gfCNCPoint3[6064] = {X 169.2391, Y 33.2115, Z -3.8333, A 0.000, B 0.000, C 0.000 }
gfCNCPoint3[6065] = {X 169.6133, Y 31.4141, Z -3.8333, A 0.000, B 0.000, C 0.000 }
gfCNCPoint3[6066] = {X 170.2096, Y 29.6777, Z -3.8333, A 0.000, B 0.000, C 0.000 }
gfCNCPoint3[6067] = {X 170.8485, Y 28.3707, Z -3.8333, A 0.000, B 0.000, C 0.000 }
gfCNCPoint3[6068] = {X 171.6564, Y 27.1608, Z -3.8333, A 0.000, B 0.000, C 0.000 }
gfCNCPoint3[6069] = {X 172.6187, Y 26.0698, Z -3.8333, A 0.000, B 0.000, C 0.000 }
gfCNCPoint3[6070] = {X 173.7182, Y 25.1171, Z -3.8333, A 0.000, B 0.000, C 0.000 }
gfCNCPoint3[6071] = {X 174.9352, Y 24.3200, Z -3.8333, A 0.000, B 0.000, C 0.000 }
gfCNCPoint3[6072] = {X 174.1525, Y 23.9324, Z -3.8333, A 0.000, B 0.000, C 0.000 }
gfCNCPoint3[6073] = {X 173.4637, Y 23.3952, Z -3.8333, A 0.000, B 0.000, C 0.000 }
gfCNCPoint3[6074] = {X 172.8971, Y 22.7305, Z -3.8333, A 0.000, B 0.000, C 0.000 }
gfCNCPoint3[6075] = {X 172.4758, Y 21.9655, Z -3.8333, A 0.000, B 0.000, C 0.000 }
gfCNCPoint3[6076] = {X 171.1581, Y 18.7388, Z -3.8333, A 0.000, B 0.000, C 0.000 }
gfCNCPoint3[6077] = {X 167.4550, Y 20.2510, Z -3.8333, A 0.000, B 0.000, C 0.000 }
gfCNCPoint3[6078] = {X 171.2322, Y 18.7085, Z -3.8333, A 0.000, B 0.000, C 0.000 }
gfCNCPoint3[6079] = {X 169.9145, Y 15.4818, Z -3.8333, A 0.000, B 0.000, C 0.000 }
gfCNCPoint3[6080] = {X 169.6699, Y 14.6462, Z -3.8333, A 0.000, B 0.000, C 0.000 }
gfCNCPoint3[6081] = {X 169.6011, Y 13.7783, Z -3.8333, A 0.000, B 0.000, C 0.000 }
gfCNCPoint3[6082] = {X 169.7111, Y 12.9146, Z -3.8333, A 0.000, B 0.000, C 0.000 }
gfCNCPoint3[6083] = {X 169.9952, Y 12.0915, Z -3.8333, A 0.000, B 0.000, C 0.000 }
gfCNCPoint3[6084] = {X 170.4414, Y 11.3439, Z -3.8333, A 0.000, B 0.000, C 0.000 }
gfCNCPoint3[6085] = {X 171.0309, Y 10.7031, Z -3.8333, A 0.000, B 0.000, C 0.000 }
gfCNCPoint3[6086] = {X 171.7389, Y 10.1963, Z -3.8333, A 0.000, B 0.000, C 0.000 }
gfCNCPoint3[6087] = {X 172.3689, Y 9.8371, Z -3.8333, A 0.000, B 0.000, C 0.000 }
gfCNCPoint3[6088] = {X 173.2427, Y 9.4701, Z -3.8333, A 0.000, B 0.000, C 0.000 }
gfCNCPoint3[6089] = {X 174.1763, Y 9.3065, Z -3.8333, A 0.000, B 0.000, C 0.000 }
gfCNCPoint3[6090] = {X 175.1229, Y 9.3543, Z -3.8333, A 0.000, B 0.000, C 0.000 }
gfCNCPoint3[6091] = {X 176.0352, Y 9.6112, Z -3.8333, A 0.000, B 0.000, C 0.000 }
gfCNCPoint3[6092] = {X 178.2247, Y 8.6863, Z -3.8333, A 0.000, B 0.000, C 0.000 }
gfCNCPoint3[6093] = {X 180.4959, Y 7.9856, Z -3.8333, A 0.000, B 0.000, C 0.000 }
gfCNCPoint3[6094] = {X 182.8259, Y 7.5163, Z -3.8333, A 0.000, B 0.000, C 0.000 }
gfCNCPoint3[6095] = {X 185.1913, Y 7.2829, Z -3.8333, A 0.000, B 0.000, C 0.000 }
gfCNCPoint3[6096] = {X 187.5681, Y 7.2880, Z -3.8333, A 0.000, B 0.000, C 0.000 }
gfCNCPoint3[6097] = {X 189.9324, Y 7.5314, Z -3.8333, A 0.000, B 0.000, C 0.000 }
gfCNCPoint3[6098] = {X 191.6817, Y 7.8911, Z -3.8333, A 0.000, B 0.000, C 0.000 }
gfCNCPoint3[6099] = {X 193.3847, Y 8.4286, Z -3.8333, A 0.000, B 0.000, C 0.000 }
gfCNCPoint3[6100] = {X 195.0236, Y 9.1381, Z -3.8333, A 0.000, B 0.000, C 0.000 }
gfCNCPoint3[6101] = {X 196.5809, Y 10.0121, Z -3.8333, A 0.000, B 0.000, C 0.000 }
gfCNCPoint3[6102] = {X 198.0403, Y 11.0414, Z -3.8333, A 0.000, B 0.000, C 0.000 }
gfCNCPoint3[6103] = {X 199.3400, Y 12.2309, Z -3.8333, A 0.000, B 0.000, C 0.000 }
gfCNCPoint3[6104] = {X 200.4666, Y 13.5854, Z -3.8333, A 0.000, B 0.000, C 0.000 }
gfCNCPoint3[6105] = {X 201.3992, Y 15.0802, Z -3.8333, A 0.000, B 0.000, C 0.000 }
gfCNCPoint3[6106] = {X 202.1206, Y 16.6876, Z -3.8333, A 0.000, B 0.000, C 0.000 }
gfCNCPoint3[6107] = {X 202.5921, Y 18.3349, Z -3.8333, A 0.000, B 0.000, C 0.000 }
gfCNCPoint3[6108] = {X 202.8719, Y 20.0254, Z -3.8333, A 0.000, B 0.000, C 0.000 }
gfCNCPoint3[6109] = {X 202.9564, Y 21.7368, Z -3.8333, A 0.000, B 0.000, C 0.000 }
gfCNCPoint3[6110] = {X 202.8443, Y 23.4466, Z -3.8333, A 0.000, B 0.000, C 0.000 }
gfCNCPoint3[6111] = {X 202.5373, Y 25.1324, Z -3.8333, A 0.000, B 0.000, C 0.000 }
gfCNCPoint3[6112] = {X 202.0878, Y 26.5970, Z -3.8333, A 0.000, B 0.000, C 0.000 }
gfCNCPoint3[6113] = {X 201.4494, Y 27.9897, Z -3.8333, A 0.000, B 0.000, C 0.000 }
gfCNCPoint3[6114] = {X 200.6332, Y 29.2862, Z -3.8333, A 0.000, B 0.000, C 0.000 }
gfCNCPoint3[6115] = {X 199.6535, Y 30.4640, Z -3.8333, A 0.000, B 0.000, C 0.000 }
gfCNCPoint3[6116] = {X 198.5272, Y 31.5026, Z -3.8333, A 0.000, B 0.000, C 0.000 }
gfCNCPoint3[6117] = {X 199.3587, Y 31.8264, Z -3.8333, A 0.000, B 0.000, C 0.000 }
gfCNCPoint3[6118] = {X 200.1039, Y 32.3172, Z -3.8333, A 0.000, B 0.000, C 0.000 }
gfCNCPoint3[6119] = {X 200.7300, Y 32.9530, Z -3.8333, A 0.000, B 0.000, C 0.000 }
gfCNCPoint3[6120] = {X 201.2091, Y 33.7058, Z -3.8333, A 0.000, B 0.000, C 0.000 }
gfCNCPoint3[6121] = {X 204.2502, Y 39.9879, Z -3.8333, A 0.000, B 0.000, C 0.000 }
gfCNCPoint3[6122] = {X 204.5648, Y 40.8802, Z -3.8333, A 0.000, B 0.000, C 0.000 }
gfCNCPoint3[6123] = {X 204.6737, Y 41.8200, Z -3.8333, A 0.000, B 0.000, C 0.000 }
gfCNCPoint3[6124] = {X 204.5715, Y 42.7606, Z -3.8333, A 0.000, B 0.000, C 0.000 }
gfCNCPoint3[6125] = {X 204.2633, Y 43.6551, Z -3.8333, A 0.000, B 0.000, C 0.000 }
gfCNCPoint3[6126] = {X 203.7643, Y 44.4590, Z -3.8333, A 0.000, B 0.000, C 0.000 }
gfCNCPoint3[6127] = {X 203.0996, Y 45.1323, Z -3.8333, A 0.000, B 0.000, C 0.000 }
gfCNCPoint3[6128] = {X 202.5633, Y 45.5658, Z -3.8333, A 0.000, B 0.000, C 0.000 }
gfCNCPoint3[6129] = {X 201.8656, Y 46.0241, Z -3.8333, A 0.000, B 0.000, C 0.000 }
gfCNCPoint3[6130] = {X 201.0918, Y 46.3373, Z -3.8333, A 0.000, B 0.000, C 0.000 }
gfCNCPoint3[6131] = {X 200.2717, Y 46.4933, Z -3.8333, A 0.000, B 0.000, C 0.000 }
gfCNCPoint3[6132] = {X 199.4370, Y 46.4861, Z -3.8333, A 0.000, B 0.000, C 0.000 }
gfCNCPoint3[6133] = {X 198.6197, Y 46.3161, Z -3.8333, A 0.000, B 0.000, C 0.000 }
gfCNCPoint3[6134] = {X 196.8802, Y 47.2412, Z -3.8333, A 0.000, B 0.000, C 0.000 }
gfCNCPoint3[6135] = {X 195.0811, Y 48.0444, Z -3.8333, A 0.000, B 0.000, C 0.000 }
gfCNCPoint3[6136] = {X 193.2311, Y 48.7221, Z -3.8333, A 0.000, B 0.000, C 0.000 }
gfCNCPoint3[6137] = {X 191.3389, Y 49.2709, Z -3.8333, A 0.000, B 0.000, C 0.000 }
gfCNCPoint3[6138] = {X 189.4027, Y 49.6631, Z -3.8333, A 0.000, B 0.000, C 0.000 }
gfCNCPoint3[6139] = {X 187.4396, Y 49.8846, Z -3.8333, A 0.000, B 0.000, C 0.000 }
gfCNCPoint3[6140] = {X 185.4646, Y 49.9336, Z -3.8333, A 0.000, B 0.000, C 0.000 }
gfCNCPoint3[6141] = {X 183.4929, Y 49.8097, Z -3.8333, A 0.000, B 0.000, C 0.000 }
gfCNCPoint3[6142] = {X 181.5396, Y 49.5138, Z -3.8333, A 0.000, B 0.000, C 0.000 }
gfCNCPoint3[6143] = {X 179.6619, Y 49.0445, Z -3.8333, A 0.000, B 0.000, C 0.000 }
gfCNCPoint3[6144] = {X 177.8500, Y 48.3642, Z -3.8333, A 0.000, B 0.000, C 0.000 }
gfCNCPoint3[6145] = {X 176.1273, Y 47.4818, Z -3.8333, A 0.000, B 0.000, C 0.000 }
gfCNCPoint3[6146] = {X 174.5165, Y 46.4089, Z -3.8333, A 0.000, B 0.000, C 0.000 }
gfCNCPoint3[6147] = {X 173.2910, Y 45.3745, Z -3.8333, A 0.000, B 0.000, C 0.000 }
gfCNCPoint3[6148] = {X 172.2004, Y 44.1988, Z -3.8333, A 0.000, B 0.000, C 0.000 }
gfCNCPoint3[6149] = {X 171.2610, Y 42.8990, Z -3.8333, A 0.000, B 0.000, C 0.000 }
gfCNCPoint3[6150] = {X 170.4868, Y 41.4946, Z -3.8333, A 0.000, B 0.000, C 0.000 }
gfCNCPoint3[6151] = {X 169.8892, Y 40.0065, Z -3.8333, A 0.000, B 0.000, C 0.000 }
gfCNCPoint3[6152] = {X 169.4771, Y 38.4567, Z -3.8333, A 0.000, B 0.000, C 0.000 }
gfCNCPoint3[6153] = {X 169.2566, Y 36.8682, Z -3.8333, A 0.000, B 0.000, C 0.000 }
gfCNCPoint3[6154] = {X 169.1729, Y 35.0439, Z -3.8333, A 0.000, B 0.000, C 0.000 }
gfCNCPoint3[6155] = {X 169.3183, Y 33.2234, Z -3.8333, A 0.000, B 0.000, C 0.000 }
gfCNCPoint3[6156] = {X 169.6904, Y 31.4354, Z -3.8333, A 0.000, B 0.000, C 0.000 }
gfCNCPoint3[6157] = {X 170.2836, Y 29.7081, Z -3.8333, A 0.000, B 0.000, C 0.000 }
gfCNCPoint3[6158] = {X 170.9356, Y 28.3799, Z -3.8333, A 0.000, B 0.000, C 0.000 }
gfCNCPoint3[6159] = {X 171.7633, Y 27.1534, Z -3.8333, A 0.000, B 0.000, C 0.000 }
gfCNCPoint3[6160] = {X 172.7511, Y 26.0519, Z -3.8333, A 0.000, B 0.000, C 0.000 }
gfCNCPoint3[6161] = {X 173.8805, Y 25.0960, Z -3.8333, A 0.000, B 0.000, C 0.000 }
gfCNCPoint3[6162] = {X 175.1302, Y 24.3037, Z -3.8333, A 0.000, B 0.000, C 0.000 }
gfCNCPoint3[6163] = {X 174.3086, Y 23.9335, Z -3.8333, A 0.000, B 0.000, C 0.000 }
gfCNCPoint3[6164] = {X 173.5838, Y 23.3981, Z -3.8333, A 0.000, B 0.000, C 0.000 }
gfCNCPoint3[6165] = {X 172.9885, Y 22.7217, Z -3.8333, A 0.000, B 0.000, C 0.000 }
gfCNCPoint3[6166] = {X 172.5496, Y 21.9347, Z -3.8333, A 0.000, B 0.000, C 0.000 }
gfCNCPoint3[6167] = {X 171.2322, Y 18.7085, Z -3.8333, A 0.000, B 0.000, C 0.000 }
gfCNCPoint3[6168] = {X 167.5291, Y 20.2207, Z -3.8333, A 0.000, B 0.000, C 0.000 }
gfCNCPoint3[6169] = {X 171.3062, Y 18.6783, Z -3.8333, A 0.000, B 0.000, C 0.000 }
gfCNCPoint3[6170] = {X 169.9886, Y 15.4516, Z -3.8333, A 0.000, B 0.000, C 0.000 }
gfCNCPoint3[6171] = {X 169.7252, Y 14.4911, Z -3.8333, A 0.000, B 0.000, C 0.000 }
gfCNCPoint3[6172] = {X 169.6977, Y 13.4955, Z -3.8333, A 0.000, B 0.000, C 0.000 }
gfCNCPoint3[6173] = {X 169.9076, Y 12.5218, Z -3.8333, A 0.000, B 0.000, C 0.000 }
gfCNCPoint3[6174] = {X 170.3429, Y 11.6260, Z -3.8333, A 0.000, B 0.000, C 0.000 }
gfCNCPoint3[6175] = {X 170.9787, Y 10.8594, Z -3.8333, A 0.000, B 0.000, C 0.000 }
gfCNCPoint3[6176] = {X 171.7785, Y 10.2658, Z -3.8333, A 0.000, B 0.000, C 0.000 }
gfCNCPoint3[6177] = {X 172.4082, Y 9.9068, Z -3.8333, A 0.000, B 0.000, C 0.000 }
gfCNCPoint3[6178] = {X 173.2740, Y 9.5443, Z -3.8333, A 0.000, B 0.000, C 0.000 }
gfCNCPoint3[6179] = {X 174.1991, Y 9.3853, Z -3.8333, A 0.000, B 0.000, C 0.000 }
gfCNCPoint3[6180] = {X 175.1362, Y 9.4376, Z -3.8333, A 0.000, B 0.000, C 0.000 }
gfCNCPoint3[6181] = {X 176.0378, Y 9.6988, Z -3.8333, A 0.000, B 0.000, C 0.000 }
gfCNCPoint3[6182] = {X 178.2241, Y 8.7716, Z -3.8333, A 0.000, B 0.000, C 0.000 }
gfCNCPoint3[6183] = {X 180.4925, Y 8.0690, Z -3.8333, A 0.000, B 0.000, C 0.000 }
gfCNCPoint3[6184] = {X 182.8201, Y 7.5980, Z -3.8333, A 0.000, B 0.000, C 0.000 }
gfCNCPoint3[6185] = {X 185.1832, Y 7.3634, Z -3.8333, A 0.000, B 0.000, C 0.000 }
gfCNCPoint3[6186] = {X 187.5580, Y 7.3676, Z -3.8333, A 0.000, B 0.000, C 0.000 }
gfCNCPoint3[6187] = {X 189.9203, Y 7.6105, Z -3.8333, A 0.000, B 0.000, C 0.000 }
gfCNCPoint3[6188] = {X 191.6615, Y 7.9685, Z -3.8333, A 0.000, B 0.000, C 0.000 }
gfCNCPoint3[6189] = {X 193.3567, Y 8.5035, Z -3.8333, A 0.000, B 0.000, C 0.000 }
gfCNCPoint3[6190] = {X 194.9880, Y 9.2097, Z -3.8333, A 0.000, B 0.000, C 0.000 }
gfCNCPoint3[6191] = {X 196.5382, Y 10.0797, Z -3.8333, A 0.000, B 0.000, C 0.000 }
gfCNCPoint3[6192] = {X 197.9908, Y 11.1044, Z -3.8333, A 0.000, B 0.000, C 0.000 }
gfCNCPoint3[6193] = {X 199.2823, Y 12.2863, Z -3.8333, A 0.000, B 0.000, C 0.000 }
gfCNCPoint3[6194] = {X 200.4017, Y 13.6323, Z -3.8333, A 0.000, B 0.000, C 0.000 }
gfCNCPoint3[6195] = {X 201.3284, Y 15.1175, Z -3.8333, A 0.000, B 0.000, C 0.000 }
gfCNCPoint3[6196] = {X 202.0453, Y 16.7146, Z -3.8333, A 0.000, B 0.000, C 0.000 }
gfCNCPoint3[6197] = {X 202.5142, Y 18.3531, Z -3.8333, A 0.000, B 0.000, C 0.000 }
gfCNCPoint3[6198] = {X 202.7924, Y 20.0344, Z -3.8333, A 0.000, B 0.000, C 0.000 }
gfCNCPoint3[6199] = {X 202.8764, Y 21.7366, Z -3.8333, A 0.000, B 0.000, C 0.000 }
gfCNCPoint3[6200] = {X 202.7649, Y 23.4371, Z -3.8333, A 0.000, B 0.000, C 0.000 }
gfCNCPoint3[6201] = {X 202.4595, Y 25.1138, Z -3.8333, A 0.000, B 0.000, C 0.000 }
gfCNCPoint3[6202] = {X 202.0016, Y 26.5984, Z -3.8333, A 0.000, B 0.000, C 0.000 }
gfCNCPoint3[6203] = {X 201.3483, Y 28.0081, Z -3.8333, A 0.000, B 0.000, C 0.000 }
gfCNCPoint3[6204] = {X 200.5114, Y 29.3171, Z -3.8333, A 0.000, B 0.000, C 0.000 }
gfCNCPoint3[6205] = {X 199.5062, Y 30.5018, Z -3.8333, A 0.000, B 0.000, C 0.000 }
gfCNCPoint3[6206] = {X 198.3508, Y 31.5406, Z -3.8333, A 0.000, B 0.000, C 0.000 }
gfCNCPoint3[6207] = {X 199.2144, Y 31.8439, Z -3.8333, A 0.000, B 0.000, C 0.000 }
gfCNCPoint3[6208] = {X 199.9908, Y 32.3287, Z -3.8333, A 0.000, B 0.000, C 0.000 }
gfCNCPoint3[6209] = {X 200.6423, Y 32.9716, Z -3.8333, A 0.000, B 0.000, C 0.000 }
gfCNCPoint3[6210] = {X 201.1375, Y 33.7414, Z -3.8333, A 0.000, B 0.000, C 0.000 }
gfCNCPoint3[6211] = {X 204.1781, Y 40.0227, Z -3.8333, A 0.000, B 0.000, C 0.000 }
gfCNCPoint3[6212] = {X 204.4868, Y 40.8982, Z -3.8333, A 0.000, B 0.000, C 0.000 }
gfCNCPoint3[6213] = {X 204.5937, Y 41.8203, Z -3.8333, A 0.000, B 0.000, C 0.000 }
gfCNCPoint3[6214] = {X 204.4934, Y 42.7431, Z -3.8333, A 0.000, B 0.000, C 0.000 }
gfCNCPoint3[6215] = {X 204.1910, Y 43.6208, Z -3.8333, A 0.000, B 0.000, C 0.000 }
gfCNCPoint3[6216] = {X 203.7015, Y 44.4095, Z -3.8333, A 0.000, B 0.000, C 0.000 }
gfCNCPoint3[6217] = {X 203.0493, Y 45.0700, Z -3.8333, A 0.000, B 0.000, C 0.000 }
gfCNCPoint3[6218] = {X 202.5131, Y 45.5036, Z -3.8333, A 0.000, B 0.000, C 0.000 }
gfCNCPoint3[6219] = {X 201.8223, Y 45.9565, Z -3.8333, A 0.000, B 0.000, C 0.000 }
gfCNCPoint3[6220] = {X 201.0558, Y 46.2645, Z -3.8333, A 0.000, B 0.000, C 0.000 }
gfCNCPoint3[6221] = {X 200.2436, Y 46.4154, Z -3.8333, A 0.000, B 0.000, C 0.000 }
gfCNCPoint3[6222] = {X 199.4177, Y 46.4035, Z -3.8333, A 0.000, B 0.000, C 0.000 }
gfCNCPoint3[6223] = {X 198.6103, Y 46.2291, Z -3.8333, A 0.000, B 0.000, C 0.000 }
gfCNCPoint3[6224] = {X 196.8688, Y 47.1577, Z -3.8333, A 0.000, B 0.000, C 0.000 }
gfCNCPoint3[6225] = {X 195.0674, Y 47.9637, Z -3.8333, A 0.000, B 0.000, C 0.000 }
gfCNCPoint3[6226] = {X 193.2146, Y 48.6433, Z -3.8333, A 0.000, B 0.000, C 0.000 }
gfCNCPoint3[6227] = {X 191.3193, Y 49.1933, Z -3.8333, A 0.000, B 0.000, C 0.000 }
gfCNCPoint3[6228] = {X 189.3899, Y 49.5842, Z -3.8333, A 0.000, B 0.000, C 0.000 }
gfCNCPoint3[6229] = {X 187.4338, Y 49.8048, Z -3.8333, A 0.000, B 0.000, C 0.000 }
gfCNCPoint3[6230] = {X 185.4659, Y 49.8536, Z -3.8333, A 0.000, B 0.000, C 0.000 }
gfCNCPoint3[6231] = {X 183.5012, Y 49.7301, Z -3.8333, A 0.000, B 0.000, C 0.000 }
gfCNCPoint3[6232] = {X 181.5549, Y 49.4353, Z -3.8333, A 0.000, B 0.000, C 0.000 }
gfCNCPoint3[6233] = {X 179.6859, Y 48.9682, Z -3.8333, A 0.000, B 0.000, C 0.000 }
gfCNCPoint3[6234] = {X 177.8824, Y 48.2911, Z -3.8333, A 0.000, B 0.000, C 0.000 }
gfCNCPoint3[6235] = {X 176.1678, Y 47.4128, Z -3.8333, A 0.000, B 0.000, C 0.000 }
gfCNCPoint3[6236] = {X 174.5644, Y 46.3449, Z -3.8333, A 0.000, B 0.000, C 0.000 }
gfCNCPoint3[6237] = {X 173.3462, Y 45.3167, Z -3.8333, A 0.000, B 0.000, C 0.000 }
gfCNCPoint3[6238] = {X 172.2622, Y 44.1479, Z -3.8333, A 0.000, B 0.000, C 0.000 }
gfCNCPoint3[6239] = {X 171.3284, Y 42.8559, Z -3.8333, A 0.000, B 0.000, C 0.000 }
gfCNCPoint3[6240] = {X 170.5588, Y 41.4598, Z -3.8333, A 0.000, B 0.000, C 0.000 }
gfCNCPoint3[6241] = {X 169.9648, Y 39.9804, Z -3.8333, A 0.000, B 0.000, C 0.000 }
gfCNCPoint3[6242] = {X 169.5553, Y 38.4398, Z -3.8333, A 0.000, B 0.000, C 0.000 }
gfCNCPoint3[6243] = {X 169.3363, Y 36.8608, Z -3.8333, A 0.000, B 0.000, C 0.000 }
gfCNCPoint3[6244] = {X 169.2528, Y 35.0461, Z -3.8333, A 0.000, B 0.000, C 0.000 }
gfCNCPoint3[6245] = {X 169.3974, Y 33.2352, Z -3.8333, A 0.000, B 0.000, C 0.000 }
gfCNCPoint3[6246] = {X 169.7675, Y 31.4567, Z -3.8333, A 0.000, B 0.000, C 0.000 }
gfCNCPoint3[6247] = {X 170.3575, Y 29.7386, Z -3.8333, A 0.000, B 0.000, C 0.000 }
gfCNCPoint3[6248] = {X 171.0242, Y 28.3867, Z -3.8333, A 0.000, B 0.000, C 0.000 }
gfCNCPoint3[6249] = {X 171.8741, Y 27.1419, Z -3.8333, A 0.000, B 0.000, C 0.000 }
gfCNCPoint3[6250] = {X 172.8906, Y 26.0288, Z -3.8333, A 0.000, B 0.000, C 0.000 }
gfCNCPoint3[6251] = {X 174.0533, Y 25.0696, Z -3.8333, A 0.000, B 0.000, C 0.000 }
gfCNCPoint3[6252] = {X 175.3393, Y 24.2834, Z -3.8333, A 0.000, B 0.000, C 0.000 }
gfCNCPoint3[6253] = {X 174.4750, Y 23.9353, Z -3.8333, A 0.000, B 0.000, C 0.000 }
gfCNCPoint3[6254] = {X 173.7098, Y 23.4037, Z -3.8333, A 0.000, B 0.000, C 0.000 }
gfCNCPoint3[6255] = {X 173.0821, Y 22.7150, Z -3.8333, A 0.000, B 0.000, C 0.000 }
gfCNCPoint3[6256] = {X 172.6235, Y 21.9039, Z -3.8333, A 0.000, B 0.000, C 0.000 }
gfCNCPoint3[6257] = {X 171.3062, Y 18.6783, Z -3.8333, A 0.000, B 0.000, C 0.000 }
gfCNCPoint3[6258] = {X 167.6031, Y 20.1905, Z -3.8333, A 0.000, B 0.000, C 0.000 }
gfCNCPoint3[6259] = {X 171.3803, Y 18.6480, Z -3.8333, A 0.000, B 0.000, C 0.000 }
gfCNCPoint3[6260] = {X 170.0626, Y 15.4213, Z -3.8333, A 0.000, B 0.000, C 0.000 }
gfCNCPoint3[6261] = {X 169.8043, Y 14.4793, Z -3.8333, A 0.000, B 0.000, C 0.000 }
gfCNCPoint3[6262] = {X 169.7773, Y 13.5028, Z -3.8333, A 0.000, B 0.000, C 0.000 }
gfCNCPoint3[6263] = {X 169.9832, Y 12.5479, Z -3.8333, A 0.000, B 0.000, C 0.000 }
gfCNCPoint3[6264] = {X 170.4102, Y 11.6694, Z -3.8333, A 0.000, B 0.000, C 0.000 }
gfCNCPoint3[6265] = {X 171.0337, Y 10.9174, Z -3.8333, A 0.000, B 0.000, C 0.000 }
gfCNCPoint3[6266] = {X 171.8181, Y 10.3353, Z -3.8333, A 0.000, B 0.000, C 0.000 }
gfCNCPoint3[6267] = {X 172.4475, Y 9.9764, Z -3.8333, A 0.000, B 0.000, C 0.000 }
gfCNCPoint3[6268] = {X 173.3053, Y 9.6186, Z -3.8333, A 0.000, B 0.000, C 0.000 }
gfCNCPoint3[6269] = {X 174.2218, Y 9.4641, Z -3.8333, A 0.000, B 0.000, C 0.000 }
gfCNCPoint3[6270] = {X 175.1494, Y 9.5211, Z -3.8333, A 0.000, B 0.000, C 0.000 }
gfCNCPoint3[6271] = {X 176.0401, Y 9.7866, Z -3.8333, A 0.000, B 0.000, C 0.000 }
gfCNCPoint3[6272] = {X 178.2232, Y 8.8572, Z -3.8333, A 0.000, B 0.000, C 0.000 }
gfCNCPoint3[6273] = {X 180.4889, Y 8.1525, Z -3.8333, A 0.000, B 0.000, C 0.000 }
gfCNCPoint3[6274] = {X 182.8141, Y 7.6798, Z -3.8333, A 0.000, B 0.000, C 0.000 }
gfCNCPoint3[6275] = {X 185.1750, Y 7.4439, Z -3.8333, A 0.000, B 0.000, C 0.000 }
gfCNCPoint3[6276] = {X 187.5478, Y 7.4472, Z -3.8333, A 0.000, B 0.000, C 0.000 }
gfCNCPoint3[6277] = {X 189.9081, Y 7.6895, Z -3.8333, A 0.000, B 0.000, C 0.000 }
gfCNCPoint3[6278] = {X 191.6413, Y 8.0459, Z -3.8333, A 0.000, B 0.000, C 0.000 }
gfCNCPoint3[6279] = {X 193.3287, Y 8.5784, Z -3.8333, A 0.000, B 0.000, C 0.000 }
gfCNCPoint3[6280] = {X 194.9525, Y 9.2814, Z -3.8333, A 0.000, B 0.000, C 0.000 }
gfCNCPoint3[6281] = {X 196.4955, Y 10.1474, Z -3.8333, A 0.000, B 0.000, C 0.000 }
gfCNCPoint3[6282] = {X 197.9414, Y 11.1673, Z -3.8333, A 0.000, B 0.000, C 0.000 }
gfCNCPoint3[6283] = {X 199.2246, Y 12.3417, Z -3.8333, A 0.000, B 0.000, C 0.000 }
gfCNCPoint3[6284] = {X 200.3368, Y 13.6791, Z -3.8333, A 0.000, B 0.000, C 0.000 }
gfCNCPoint3[6285] = {X 201.2577, Y 15.1548, Z -3.8333, A 0.000, B 0.000, C 0.000 }
gfCNCPoint3[6286] = {X 201.9701, Y 16.7417, Z -3.8333, A 0.000, B 0.000, C 0.000 }
gfCNCPoint3[6287] = {X 202.4363, Y 18.3712, Z -3.8333, A 0.000, B 0.000, C 0.000 }
gfCNCPoint3[6288] = {X 202.7129, Y 20.0435, Z -3.8333, A 0.000, B 0.000, C 0.000 }
gfCNCPoint3[6289] = {X 202.7964, Y 21.7363, Z -3.8333, A 0.000, B 0.000, C 0.000 }
gfCNCPoint3[6290] = {X 202.6855, Y 23.4277, Z -3.8333, A 0.000, B 0.000, C 0.000 }
gfCNCPoint3[6291] = {X 202.3817, Y 25.0952, Z -3.8333, A 0.000, B 0.000, C 0.000 }
gfCNCPoint3[6292] = {X 201.9145, Y 26.6019, Z -3.8333, A 0.000, B 0.000, C 0.000 }
gfCNCPoint3[6293] = {X 201.2448, Y 28.0301, Z -3.8333, A 0.000, B 0.000, C 0.000 }
gfCNCPoint3[6294] = {X 200.3851, Y 29.3527, Z -3.8333, A 0.000, B 0.000, C 0.000 }
gfCNCPoint3[6295] = {X 199.3518, Y 30.5447, Z -3.8333, A 0.000, B 0.000, C 0.000 }
gfCNCPoint3[6296] = {X 198.1646, Y 31.5833, Z -3.8333, A 0.000, B 0.000, C 0.000 }
gfCNCPoint3[6297] = {X 199.0626, Y 31.8620, Z -3.8333, A 0.000, B 0.000, C 0.000 }
gfCNCPoint3[6298] = {X 199.8730, Y 32.3388, Z -3.8333, A 0.000, B 0.000, C 0.000 }
gfCNCPoint3[6299] = {X 200.5528, Y 32.9886, Z -3.8333, A 0.000, B 0.000, C 0.000 }
gfCNCPoint3[6300] = {X 201.0657, Y 33.7766, Z -3.8333, A 0.000, B 0.000, C 0.000 }
gfCNCPoint3[6301] = {X 204.1061, Y 40.0576, Z -3.8333, A 0.000, B 0.000, C 0.000 }
gfCNCPoint3[6302] = {X 204.4089, Y 40.9162, Z -3.8333, A 0.000, B 0.000, C 0.000 }
gfCNCPoint3[6303] = {X 204.5137, Y 41.8206, Z -3.8333, A 0.000, B 0.000, C 0.000 }
gfCNCPoint3[6304] = {X 204.4154, Y 42.7257, Z -3.8333, A 0.000, B 0.000, C 0.000 }
gfCNCPoint3[6305] = {X 204.1188, Y 43.5864, Z -3.8333, A 0.000, B 0.000, C 0.000 }
gfCNCPoint3[6306] = {X 203.6387, Y 44.3600, Z -3.8333, A 0.000, B 0.000, C 0.000 }
gfCNCPoint3[6307] = {X 202.9990, Y 45.0078, Z -3.8333, A 0.000, B 0.000, C 0.000 }
gfCNCPoint3[6308] = {X 202.4628, Y 45.4414, Z -3.8333, A 0.000, B 0.000, C 0.000 }
gfCNCPoint3[6309] = {X 201.7789, Y 45.8889, Z -3.8333, A 0.000, B 0.000, C 0.000 }
gfCNCPoint3[6310] = {X 201.0198, Y 46.1916, Z -3.8333, A 0.000, B 0.000, C 0.000 }
gfCNCPoint3[6311] = {X 200.2157, Y 46.3375, Z -3.8333, A 0.000, B 0.000, C 0.000 }
gfCNCPoint3[6312] = {X 199.3986, Y 46.3207, Z -3.8333, A 0.000, B 0.000, C 0.000 }
gfCNCPoint3[6313] = {X 198.6011, Y 46.1420, Z -3.8333, A 0.000, B 0.000, C 0.000 }
gfCNCPoint3[6314] = {X 196.8577, Y 47.0740, Z -3.8333, A 0.000, B 0.000, C 0.000 }
gfCNCPoint3[6315] = {X 195.0538, Y 47.8828, Z -3.8333, A 0.000, B 0.000, C 0.000 }
gfCNCPoint3[6316] = {X 193.1981, Y 48.5645, Z -3.8333, A 0.000, B 0.000, C 0.000 }
gfCNCPoint3[6317] = {X 191.2996, Y 49.1157, Z -3.8333, A 0.000, B 0.000, C 0.000 }
gfCNCPoint3[6318] = {X 189.3772, Y 49.5052, Z -3.8333, A 0.000, B 0.000, C 0.000 }
gfCNCPoint3[6319] = {X 187.4280, Y 49.7250, Z -3.8333, A 0.000, B 0.000, C 0.000 }
gfCNCPoint3[6320] = {X 185.4671, Y 49.7736, Z -3.8333, A 0.000, B 0.000, C 0.000 }
gfCNCPoint3[6321] = {X 183.5094, Y 49.6505, Z -3.8333, A 0.000, B 0.000, C 0.000 }
gfCNCPoint3[6322] = {X 181.5701, Y 49.3567, Z -3.8333, A 0.000, B 0.000, C 0.000 }
gfCNCPoint3[6323] = {X 179.7099, Y 48.8918, Z -3.8333, A 0.000, B 0.000, C 0.000 }
gfCNCPoint3[6324] = {X 177.9148, Y 48.2179, Z -3.8333, A 0.000, B 0.000, C 0.000 }
gfCNCPoint3[6325] = {X 176.2082, Y 47.3438, Z -3.8333, A 0.000, B 0.000, C 0.000 }
gfCNCPoint3[6326] = {X 174.6124, Y 46.2809, Z -3.8333, A 0.000, B 0.000, C 0.000 }
gfCNCPoint3[6327] = {X 173.4015, Y 45.2588, Z -3.8333, A 0.000, B 0.000, C 0.000 }
gfCNCPoint3[6328] = {X 172.3239, Y 44.0970, Z -3.8333, A 0.000, B 0.000, C 0.000 }
gfCNCPoint3[6329] = {X 171.3958, Y 42.8127, Z -3.8333, A 0.000, B 0.000, C 0.000 }
gfCNCPoint3[6330] = {X 170.6308, Y 41.4249, Z -3.8333, A 0.000, B 0.000, C 0.000 }
gfCNCPoint3[6331] = {X 170.0405, Y 39.9544, Z -3.8333, A 0.000, B 0.000, C 0.000 }
gfCNCPoint3[6332] = {X 169.6335, Y 38.4230, Z -3.8333, A 0.000, B 0.000, C 0.000 }
gfCNCPoint3[6333] = {X 169.4159, Y 36.8534, Z -3.8333, A 0.000, B 0.000, C 0.000 }
gfCNCPoint3[6334] = {X 169.3328, Y 35.0483, Z -3.8333, A 0.000, B 0.000, C 0.000 }
gfCNCPoint3[6335] = {X 169.4765, Y 33.2471, Z -3.8333, A 0.000, B 0.000, C 0.000 }
gfCNCPoint3[6336] = {X 169.8447, Y 31.4780, Z -3.8333, A 0.000, B 0.000, C 0.000 }
gfCNCPoint3[6337] = {X 170.4315, Y 29.7690, Z -3.8333, A 0.000, B 0.000, C 0.000 }
gfCNCPoint3[6338] = {X 171.1148, Y 28.3902, Z -3.8333, A 0.000, B 0.000, C 0.000 }
gfCNCPoint3[6339] = {X 171.9902, Y 27.1247, Z -3.8333, A 0.000, B 0.000, C 0.000 }
gfCNCPoint3[6340] = {X 173.0392, Y 25.9989, Z -3.8333, A 0.000, B 0.000, C 0.000 }
gfCNCPoint3[6341] = {X 174.2400, Y 25.0365, Z -3.8333, A 0.000, B 0.000, C 0.000 }
gfCNCPoint3[6342] = {X 175.5672, Y 24.2578, Z -3.8333, A 0.000, B 0.000, C 0.000 }
gfCNCPoint3[6343] = {X 174.6550, Y 23.9381, Z -3.8333, A 0.000, B 0.000, C 0.000 }
gfCNCPoint3[6344] = {X 173.8437, Y 23.4127, Z -3.8333, A 0.000, B 0.000, C 0.000 }
gfCNCPoint3[6345] = {X 173.1787, Y 22.7113, Z -3.8333, A 0.000, B 0.000, C 0.000 }
gfCNCPoint3[6346] = {X 172.6973, Y 21.8731, Z -3.8333, A 0.000, B 0.000, C 0.000 }
gfCNCPoint3[6347] = {X 171.3803, Y 18.6480, Z -3.8333, A 0.000, B 0.000, C 0.000 }
gfCNCPoint3[6348] = {X 167.6770, Y 20.1603, Z -3.8333, A 0.000, B 0.000, C 0.000 }
gfCNCPoint3[6349] = {X 167.6769, Y 20.1601, Z -3.8333, A 0.000, B 0.000, C 0.000 }
gfCNCPoint3[6350] = {X 171.4542, Y 18.6179, Z -3.8333, A 0.000, B 0.000, C 0.000 }
gfCNCPoint3[6351] = {X 170.1367, Y 15.3911, Z -3.8333, A 0.000, B 0.000, C 0.000 }
gfCNCPoint3[6352] = {X 169.8835, Y 14.4675, Z -3.8333, A 0.000, B 0.000, C 0.000 }
gfCNCPoint3[6353] = {X 169.8570, Y 13.5102, Z -3.8333, A 0.000, B 0.000, C 0.000 }
gfCNCPoint3[6354] = {X 170.0588, Y 12.5740, Z -3.8333, A 0.000, B 0.000, C 0.000 }
gfCNCPoint3[6355] = {X 170.4774, Y 11.7127, Z -3.8333, A 0.000, B 0.000, C 0.000 }
gfCNCPoint3[6356] = {X 171.0888, Y 10.9755, Z -3.8333, A 0.000, B 0.000, C 0.000 }
gfCNCPoint3[6357] = {X 171.8578, Y 10.4048, Z -3.8333, A 0.000, B 0.000, C 0.000 }
gfCNCPoint3[6358] = {X 172.4867, Y 10.0462, Z -3.8333, A 0.000, B 0.000, C 0.000 }
gfCNCPoint3[6359] = {X 173.3363, Y 9.6929, Z -3.8333, A 0.000, B 0.000, C 0.000 }
gfCNCPoint3[6360] = {X 174.2443, Y 9.5431, Z -3.8333, A 0.000, B 0.000, C 0.000 }
gfCNCPoint3[6361] = {X 175.1624, Y 9.6048, Z -3.8333, A 0.000, B 0.000, C 0.000 }
gfCNCPoint3[6362] = {X 176.0421, Y 9.8746, Z -3.8333, A 0.000, B 0.000, C 0.000 }
gfCNCPoint3[6363] = {X 177.9051, Y 9.0624, Z -3.8333, A 0.000, B 0.000, C 0.000 }
gfCNCPoint3[6364] = {X 179.8314, Y 8.4146, Z -3.8333, A 0.000, B 0.000, C 0.000 }
gfCNCPoint3[6365] = {X 181.8066, Y 7.9362, Z -3.8333, A 0.000, B 0.000, C 0.000 }
gfCNCPoint3[6366] = {X 183.8158, Y 7.6308, Z -3.8333, A 0.000, B 0.000, C 0.000 }
gfCNCPoint3[6367] = {X 185.8440, Y 7.5006, Z -3.8333, A 0.000, B 0.000, C 0.000 }
gfCNCPoint3[6368] = {X 187.8758, Y 7.5467, Z -3.8333, A 0.000, B 0.000, C 0.000 }
gfCNCPoint3[6369] = {X 189.8959, Y 7.7686, Z -3.8333, A 0.000, B 0.000, C 0.000 }
gfCNCPoint3[6370] = {X 191.6211, Y 8.1233, Z -3.8333, A 0.000, B 0.000, C 0.000 }
gfCNCPoint3[6371] = {X 193.3006, Y 8.6533, Z -3.8333, A 0.000, B 0.000, C 0.000 }
gfCNCPoint3[6372] = {X 194.9169, Y 9.3530, Z -3.8333, A 0.000, B 0.000, C 0.000 }
gfCNCPoint3[6373] = {X 196.4528, Y 10.2150, Z -3.8333, A 0.000, B 0.000, C 0.000 }
gfCNCPoint3[6374] = {X 197.8920, Y 11.2302, Z -3.8333, A 0.000, B 0.000, C 0.000 }
gfCNCPoint3[6375] = {X 199.1669, Y 12.3971, Z -3.8333, A 0.000, B 0.000, C 0.000 }
gfCNCPoint3[6376] = {X 200.2720, Y 13.7259, Z -3.8333, A 0.000, B 0.000, C 0.000 }
gfCNCPoint3[6377] = {X 201.1869, Y 15.1921, Z -3.8333, A 0.000, B 0.000, C 0.000 }
gfCNCPoint3[6378] = {X 201.8948, Y 16.7687, Z -3.8333, A 0.000, B 0.000, C 0.000 }
gfCNCPoint3[6379] = {X 202.3584, Y 18.3894, Z -3.8333, A 0.000, B 0.000, C 0.000 }
gfCNCPoint3[6380] = {X 202.6334, Y 20.0525, Z -3.8333, A 0.000, B 0.000, C 0.000 }
gfCNCPoint3[6381] = {X 202.7164, Y 21.7361, Z -3.8333, A 0.000, B 0.000, C 0.000 }
gfCNCPoint3[6382] = {X 202.6060, Y 23.4182, Z -3.8333, A 0.000, B 0.000, C 0.000 }
gfCNCPoint3[6383] = {X 202.3039, Y 25.0766, Z -3.8333, A 0.000, B 0.000, C 0.000 }
gfCNCPoint3[6384] = {X 201.8264, Y 26.6077, Z -3.8333, A 0.000, B 0.000, C 0.000 }
gfCNCPoint3[6385] = {X 201.1382, Y 28.0565, Z -3.8333, A 0.000, B 0.000, C 0.000 }
gfCNCPoint3[6386] = {X 200.2531, Y 29.3941, Z -3.8333, A 0.000, B 0.000, C 0.000 }
gfCNCPoint3[6387] = {X 199.1886, Y 30.5938, Z -3.8333, A 0.000, B 0.000, C 0.000 }
gfCNCPoint3[6388] = {X 197.9659, Y 31.6319, Z -3.8333, A 0.000, B 0.000, C 0.000 }
gfCNCPoint3[6389] = {X 198.7277, Y 31.8158, Z -3.8333, A 0.000, B 0.000, C 0.000 }
gfCNCPoint3[6390] = {X 199.4391, Y 32.1448, Z -3.8333, A 0.000, B 0.000, C 0.000 }
gfCNCPoint3[6391] = {X 200.0726, Y 32.6061, Z -3.8333, A 0.000, B 0.000, C 0.000 }
gfCNCPoint3[6392] = {X 200.6040, Y 33.1821, Z -3.8333, A 0.000, B 0.000, C 0.000 }
gfCNCPoint3[6393] = {X 201.0129, Y 33.8507, Z -3.8333, A 0.000, B 0.000, C 0.000 }
gfCNCPoint3[6394] = {X 204.0341, Y 40.0925, Z -3.8333, A 0.000, B 0.000, C 0.000 }
gfCNCPoint3[6395] = {X 204.3309, Y 40.9342, Z -3.8333, A 0.000, B 0.000, C 0.000 }
gfCNCPoint3[6396] = {X 204.4337, Y 41.8209, Z -3.8333, A 0.000, B 0.000, C 0.000 }
gfCNCPoint3[6397] = {X 204.3373, Y 42.7082, Z -3.8333, A 0.000, B 0.000, C 0.000 }
gfCNCPoint3[6398] = {X 204.0465, Y 43.5521, Z -3.8333, A 0.000, B 0.000, C 0.000 }
gfCNCPoint3[6399] = {X 203.5758, Y 44.3105, Z -3.8333, A 0.000, B 0.000, C 0.000 }
gfCNCPoint3[6400] = {X 202.9487, Y 44.9456, Z -3.8333, A 0.000, B 0.000, C 0.000 }
gfCNCPoint3[6401] = {X 202.4125, Y 45.3791, Z -3.8333, A 0.000, B 0.000, C 0.000 }
gfCNCPoint3[6402] = {X 201.7357, Y 45.8212, Z -3.8333, A 0.000, B 0.000, C 0.000 }
gfCNCPoint3[6403] = {X 200.9839, Y 46.1186, Z -3.8333, A 0.000, B 0.000, C 0.000 }
gfCNCPoint3[6404] = {X 200.1879, Y 46.2594, Z -3.8333, A 0.000, B 0.000, C 0.000 }
gfCNCPoint3[6405] = {X 199.3797, Y 46.2377, Z -3.8333, A 0.000, B 0.000, C 0.000 }
gfCNCPoint3[6406] = {X 198.5923, Y 46.0546, Z -3.8333, A 0.000, B 0.000, C 0.000 }
gfCNCPoint3[6407] = {X 196.8468, Y 46.9902, Z -3.8333, A 0.000, B 0.000, C 0.000 }
gfCNCPoint3[6408] = {X 195.0404, Y 47.8019, Z -3.8333, A 0.000, B 0.000, C 0.000 }
gfCNCPoint3[6409] = {X 193.1818, Y 48.4857, Z -3.8333, A 0.000, B 0.000, C 0.000 }
gfCNCPoint3[6410] = {X 191.2800, Y 49.0382, Z -3.8333, A 0.000, B 0.000, C 0.000 }
gfCNCPoint3[6411] = {X 189.3644, Y 49.4262, Z -3.8333, A 0.000, B 0.000, C 0.000 }
gfCNCPoint3[6412] = {X 187.4222, Y 49.6453, Z -3.8333, A 0.000, B 0.000, C 0.000 }
gfCNCPoint3[6413] = {X 185.4683, Y 49.6936, Z -3.8333, A 0.000, B 0.000, C 0.000 }
gfCNCPoint3[6414] = {X 183.5177, Y 49.5710, Z -3.8333, A 0.000, B 0.000, C 0.000 }
gfCNCPoint3[6415] = {X 181.5852, Y 49.2782, Z -3.8333, A 0.000, B 0.000, C 0.000 }
gfCNCPoint3[6416] = {X 179.7338, Y 48.8155, Z -3.8333, A 0.000, B 0.000, C 0.000 }
gfCNCPoint3[6417] = {X 177.9472, Y 48.1448, Z -3.8333, A 0.000, B 0.000, C 0.000 }
gfCNCPoint3[6418] = {X 176.2487, Y 47.2748, Z -3.8333, A 0.000, B 0.000, C 0.000 }
gfCNCPoint3[6419] = {X 174.6604, Y 46.2169, Z -3.8333, A 0.000, B 0.000, C 0.000 }
gfCNCPoint3[6420] = {X 173.4567, Y 45.2010, Z -3.8333, A 0.000, B 0.000, C 0.000 }
gfCNCPoint3[6421] = {X 172.3856, Y 44.0462, Z -3.8333, A 0.000, B 0.000, C 0.000 }
gfCNCPoint3[6422] = {X 171.4631, Y 42.7695, Z -3.8333, A 0.000, B 0.000, C 0.000 }
gfCNCPoint3[6423] = {X 170.7028, Y 41.3901, Z -3.8333, A 0.000, B 0.000, C 0.000 }
gfCNCPoint3[6424] = {X 170.1161, Y 39.9284, Z -3.8333, A 0.000, B 0.000, C 0.000 }
gfCNCPoint3[6425] = {X 169.7117, Y 38.4061, Z -3.8333, A 0.000, B 0.000, C 0.000 }
gfCNCPoint3[6426] = {X 169.4956, Y 36.8460, Z -3.8333, A 0.000, B 0.000, C 0.000 }
gfCNCPoint3[6427] = {X 169.4128, Y 35.0506, Z -3.8333, A 0.000, B 0.000, C 0.000 }
gfCNCPoint3[6428] = {X 169.5556, Y 33.2589, Z -3.8333, A 0.000, B 0.000, C 0.000 }
gfCNCPoint3[6429] = {X 169.9218, Y 31.4993, Z -3.8333, A 0.000, B 0.000, C 0.000 }
gfCNCPoint3[6430] = {X 170.5055, Y 29.7995, Z -3.8333, A 0.000, B 0.000, C 0.000 }
gfCNCPoint3[6431] = {X 171.2084, Y 28.3893, Z -3.8333, A 0.000, B 0.000, C 0.000 }
gfCNCPoint3[6432] = {X 172.1136, Y 27.0997, Z -3.8333, A 0.000, B 0.000, C 0.000 }
gfCNCPoint3[6433] = {X 173.2009, Y 25.9594, Z -3.8333, A 0.000, B 0.000, C 0.000 }
gfCNCPoint3[6434] = {X 174.4461, Y 24.9939, Z -3.8333, A 0.000, B 0.000, C 0.000 }
gfCNCPoint3[6435] = {X 175.8213, Y 24.2248, Z -3.8333, A 0.000, B 0.000, C 0.000 }
gfCNCPoint3[6436] = {X 175.0303, Y 24.0138, Z -3.8333, A 0.000, B 0.000, C 0.000 }
gfCNCPoint3[6437] = {X 174.2988, Y 23.6463, Z -3.8333, A 0.000, B 0.000, C 0.000 }
gfCNCPoint3[6438] = {X 173.6575, Y 23.1375, Z -3.8333, A 0.000, B 0.000, C 0.000 }
gfCNCPoint3[6439] = {X 173.1332, Y 22.5088, Z -3.8333, A 0.000, B 0.000, C 0.000 }
gfCNCPoint3[6440] = {X 172.7479, Y 21.7866, Z -3.8333, A 0.000, B 0.000, C 0.000 }
gfCNCPoint3[6441] = {X 171.4542, Y 18.6179, Z -3.8333, A 0.000, B 0.000, C 0.000 }
gfCNCPoint3[6442] = {X 167.6769, Y 20.1601, Z -3.8333, A 0.000, B 0.000, C 0.000 }
gfCNCPoint3[6443] = {X 167.6769, Y 20.1601, Z -0.8333, A 0.000, B 0.000, C 0.000 }
gfCNCPoint3[6444] = {X 167.6769, Y 20.1601, Z 11.0000, A 0.000, B 0.000, C 0.000 }
gfCNCPoint3[6445] = {X 210.1652, Y 28.5741, Z 11.0000, A 0.000, B 0.000, C 0.000 }
gfCNCPoint3[6446] = {X 210.1652, Y 28.5741, Z -0.8333, A 0.000, B 0.000, C 0.000 }
gfCNCPoint3[6447] = {X 210.1652, Y 28.5741, Z -3.8333, A 0.000, B 0.000, C 0.000 }
gfCNCPoint3[6448] = {X 214.2452, Y 28.5741, Z -3.8333, A 0.000, B 0.000, C 0.000 }
gfCNCPoint3[6449] = {X 214.2452, Y 17.4624, Z -3.8333, A 0.000, B 0.000, C 0.000 }
gfCNCPoint3[6450] = {X 214.2399, Y 16.7693, Z -3.8333, A 0.000, B 0.000, C 0.000 }
gfCNCPoint3[6451] = {X 214.2429, Y 16.2728, Z -3.8333, A 0.000, B 0.000, C 0.000 }
gfCNCPoint3[6452] = {X 213.6049, Y 15.6016, Z -3.8333, A 0.000, B 0.000, C 0.000 }
gfCNCPoint3[6453] = {X 213.1247, Y 14.8099, Z -3.8333, A 0.000, B 0.000, C 0.000 }
gfCNCPoint3[6454] = {X 212.8241, Y 13.9341, Z -3.8333, A 0.000, B 0.000, C 0.000 }
gfCNCPoint3[6455] = {X 212.7172, Y 13.0143, Z -3.8333, A 0.000, B 0.000, C 0.000 }
gfCNCPoint3[6456] = {X 212.7170, Y 12.1868, Z -3.8333, A 0.000, B 0.000, C 0.000 }
gfCNCPoint3[6457] = {X 212.8253, Y 11.2255, Z -3.8333, A 0.000, B 0.000, C 0.000 }
gfCNCPoint3[6458] = {X 213.1448, Y 10.3124, Z -3.8333, A 0.000, B 0.000, C 0.000 }
gfCNCPoint3[6459] = {X 213.6595, Y 9.4933, Z -3.8333, A 0.000, B 0.000, C 0.000 }
gfCNCPoint3[6460] = {X 214.3435, Y 8.8093, Z -3.8333, A 0.000, B 0.000, C 0.000 }
gfCNCPoint3[6461] = {X 215.1626, Y 8.2946, Z -3.8333, A 0.000, B 0.000, C 0.000 }
gfCNCPoint3[6462] = {X 216.0757, Y 7.9751, Z -3.8333, A 0.000, B 0.000, C 0.000 }
gfCNCPoint3[6463] = {X 217.0370, Y 7.8668, Z -3.8333, A 0.000, B 0.000, C 0.000 }
gfCNCPoint3[6464] = {X 223.4805, Y 7.8668, Z -3.8333, A 0.000, B 0.000, C 0.000 }
gfCNCPoint3[6465] = {X 224.4418, Y 7.9751, Z -3.8333, A 0.000, B 0.000, C 0.000 }
gfCNCPoint3[6466] = {X 225.3549, Y 8.2946, Z -3.8333, A 0.000, B 0.000, C 0.000 }
gfCNCPoint3[6467] = {X 226.1740, Y 8.8093, Z -3.8333, A 0.000, B 0.000, C 0.000 }
gfCNCPoint3[6468] = {X 226.8580, Y 9.4933, Z -3.8333, A 0.000, B 0.000, C 0.000 }
gfCNCPoint3[6469] = {X 227.3727, Y 10.3124, Z -3.8333, A 0.000, B 0.000, C 0.000 }
gfCNCPoint3[6470] = {X 227.6922, Y 11.2255, Z -3.8333, A 0.000, B 0.000, C 0.000 }
gfCNCPoint3[6471] = {X 227.8005, Y 12.1868, Z -3.8333, A 0.000, B 0.000, C 0.000 }
gfCNCPoint3[6472] = {X 227.8005, Y 12.9781, Z -3.8333, A 0.000, B 0.000, C 0.000 }
gfCNCPoint3[6473] = {X 227.6992, Y 13.9081, Z -3.8333, A 0.000, B 0.000, C 0.000 }
gfCNCPoint3[6474] = {X 227.4000, Y 14.7945, Z -3.8333, A 0.000, B 0.000, C 0.000 }
gfCNCPoint3[6475] = {X 226.9171, Y 15.5957, Z -3.8333, A 0.000, B 0.000, C 0.000 }
gfCNCPoint3[6476] = {X 226.2729, Y 16.2742, Z -3.8333, A 0.000, B 0.000, C 0.000 }
gfCNCPoint3[6477] = {X 226.2739, Y 40.9154, Z -3.8333, A 0.000, B 0.000, C 0.000 }
gfCNCPoint3[6478] = {X 226.9113, Y 41.5855, Z -3.8333, A 0.000, B 0.000, C 0.000 }
gfCNCPoint3[6479] = {X 227.3914, Y 42.3759, Z -3.8333, A 0.000, B 0.000, C 0.000 }
gfCNCPoint3[6480] = {X 227.6924, Y 43.2504, Z -3.8333, A 0.000, B 0.000, C 0.000 }
gfCNCPoint3[6481] = {X 227.8003, Y 44.1689, Z -3.8333, A 0.000, B 0.000, C 0.000 }
gfCNCPoint3[6482] = {X 227.8005, Y 45.0000, Z -3.8333, A 0.000, B 0.000, C 0.000 }
gfCNCPoint3[6483] = {X 227.6922, Y 45.9613, Z -3.8333, A 0.000, B 0.000, C 0.000 }
gfCNCPoint3[6484] = {X 227.3727, Y 46.8744, Z -3.8333, A 0.000, B 0.000, C 0.000 }
gfCNCPoint3[6485] = {X 226.8580, Y 47.6935, Z -3.8333, A 0.000, B 0.000, C 0.000 }
gfCNCPoint3[6486] = {X 226.1740, Y 48.3775, Z -3.8333, A 0.000, B 0.000, C 0.000 }
gfCNCPoint3[6487] = {X 225.3549, Y 48.8922, Z -3.8333, A 0.000, B 0.000, C 0.000 }
gfCNCPoint3[6488] = {X 224.4418, Y 49.2117, Z -3.8333, A 0.000, B 0.000, C 0.000 }
gfCNCPoint3[6489] = {X 223.4805, Y 49.3200, Z -3.8333, A 0.000, B 0.000, C 0.000 }
gfCNCPoint3[6490] = {X 217.0370, Y 49.3200, Z -3.8333, A 0.000, B 0.000, C 0.000 }
gfCNCPoint3[6491] = {X 216.0805, Y 49.2128, Z -3.8333, A 0.000, B 0.000, C 0.000 }
gfCNCPoint3[6492] = {X 215.1715, Y 48.8964, Z -3.8333, A 0.000, B 0.000, C 0.000 }
gfCNCPoint3[6493] = {X 214.3551, Y 48.3867, Z -3.8333, A 0.000, B 0.000, C 0.000 }
gfCNCPoint3[6494] = {X 213.6718, Y 47.7088, Z -3.8333, A 0.000, B 0.000, C 0.000 }
gfCNCPoint3[6495] = {X 213.1556, Y 46.8965, Z -3.8333, A 0.000, B 0.000, C 0.000 }
gfCNCPoint3[6496] = {X 212.8320, Y 45.9901, Z -3.8333, A 0.000, B 0.000, C 0.000 }
gfCNCPoint3[6497] = {X 212.7172, Y 45.0345, Z -3.8333, A 0.000, B 0.000, C 0.000 }
gfCNCPoint3[6498] = {X 212.7170, Y 44.1967, Z -3.8333, A 0.000, B 0.000, C 0.000 }
gfCNCPoint3[6499] = {X 212.7889, Y 43.4182, Z -3.8333, A 0.000, B 0.000, C 0.000 }
gfCNCPoint3[6500] = {X 213.0020, Y 42.6661, Z -3.8333, A 0.000, B 0.000, C 0.000 }
gfCNCPoint3[6501] = {X 213.3493, Y 41.9658, Z -3.8333, A 0.000, B 0.000, C 0.000 }
gfCNCPoint3[6502] = {X 213.8189, Y 41.3408, Z -3.8333, A 0.000, B 0.000, C 0.000 }
gfCNCPoint3[6503] = {X 214.2408, Y 40.8754, Z -3.8333, A 0.000, B 0.000, C 0.000 }
gfCNCPoint3[6504] = {X 214.2452, Y 40.3062, Z -3.8333, A 0.000, B 0.000, C 0.000 }
gfCNCPoint3[6505] = {X 214.2452, Y 28.5741, Z -3.8333, A 0.000, B 0.000, C 0.000 }
gfCNCPoint3[6506] = {X 210.2452, Y 28.5741, Z -3.8333, A 0.000, B 0.000, C 0.000 }
gfCNCPoint3[6507] = {X 214.3252, Y 28.5741, Z -3.8333, A 0.000, B 0.000, C 0.000 }
gfCNCPoint3[6508] = {X 214.3252, Y 17.4621, Z -3.8333, A 0.000, B 0.000, C 0.000 }
gfCNCPoint3[6509] = {X 214.3199, Y 16.7692, Z -3.8333, A 0.000, B 0.000, C 0.000 }
gfCNCPoint3[6510] = {X 214.3231, Y 16.2357, Z -3.8333, A 0.000, B 0.000, C 0.000 }
gfCNCPoint3[6511] = {X 213.6855, Y 15.5751, Z -3.8333, A 0.000, B 0.000, C 0.000 }
gfCNCPoint3[6512] = {X 213.2050, Y 14.7928, Z -3.8333, A 0.000, B 0.000, C 0.000 }
gfCNCPoint3[6513] = {X 212.9042, Y 13.9255, Z -3.8333, A 0.000, B 0.000, C 0.000 }
gfCNCPoint3[6514] = {X 212.7972, Y 13.0136, Z -3.8333, A 0.000, B 0.000, C 0.000 }
gfCNCPoint3[6515] = {X 212.7970, Y 12.1868, Z -3.8333, A 0.000, B 0.000, C 0.000 }
gfCNCPoint3[6516] = {X 212.9033, Y 11.2433, Z -3.8333, A 0.000, B 0.000, C 0.000 }
gfCNCPoint3[6517] = {X 213.2169, Y 10.3472, Z -3.8333, A 0.000, B 0.000, C 0.000 }
gfCNCPoint3[6518] = {X 213.7220, Y 9.5432, Z -3.8333, A 0.000, B 0.000, C 0.000 }
gfCNCPoint3[6519] = {X 214.3934, Y 8.8719, Z -3.8333, A 0.000, B 0.000, C 0.000 }
gfCNCPoint3[6520] = {X 215.1973, Y 8.3667, Z -3.8333, A 0.000, B 0.000, C 0.000 }
gfCNCPoint3[6521] = {X 216.0935, Y 8.0531, Z -3.8333, A 0.000, B 0.000, C 0.000 }
gfCNCPoint3[6522] = {X 217.0370, Y 7.9468, Z -3.8333, A 0.000, B 0.000, C 0.000 }
gfCNCPoint3[6523] = {X 223.4805, Y 7.9468, Z -3.8333, A 0.000, B 0.000, C 0.000 }
gfCNCPoint3[6524] = {X 224.4240, Y 8.0531, Z -3.8333, A 0.000, B 0.000, C 0.000 }
gfCNCPoint3[6525] = {X 225.3201, Y 8.3667, Z -3.8333, A 0.000, B 0.000, C 0.000 }
gfCNCPoint3[6526] = {X 226.1241, Y 8.8718, Z -3.8333, A 0.000, B 0.000, C 0.000 }
gfCNCPoint3[6527] = {X 226.7954, Y 9.5432, Z -3.8333, A 0.000, B 0.000, C 0.000 }
gfCNCPoint3[6528] = {X 227.3006, Y 10.3471, Z -3.8333, A 0.000, B 0.000, C 0.000 }
gfCNCPoint3[6529] = {X 227.6142, Y 11.2433, Z -3.8333, A 0.000, B 0.000, C 0.000 }
gfCNCPoint3[6530] = {X 227.7205, Y 12.1868, Z -3.8333, A 0.000, B 0.000, C 0.000 }
gfCNCPoint3[6531] = {X 227.7205, Y 12.9781, Z -3.8333, A 0.000, B 0.000, C 0.000 }
gfCNCPoint3[6532] = {X 227.6190, Y 13.8999, Z -3.8333, A 0.000, B 0.000, C 0.000 }
gfCNCPoint3[6533] = {X 227.3196, Y 14.7776, Z -3.8333, A 0.000, B 0.000, C 0.000 }
gfCNCPoint3[6534] = {X 226.8366, Y 15.5692, Z -3.8333, A 0.000, B 0.000, C 0.000 }
gfCNCPoint3[6535] = {X 226.1929, Y 16.2369, Z -3.8333, A 0.000, B 0.000, C 0.000 }
gfCNCPoint3[6536] = {X 226.1939, Y 40.9527, Z -3.8333, A 0.000, B 0.000, C 0.000 }
gfCNCPoint3[6537] = {X 226.8308, Y 41.6122, Z -3.8333, A 0.000, B 0.000, C 0.000 }
gfCNCPoint3[6538] = {X 227.3111, Y 42.3932, Z -3.8333, A 0.000, B 0.000, C 0.000 }
gfCNCPoint3[6539] = {X 227.6123, Y 43.2592, Z -3.8333, A 0.000, B 0.000, C 0.000 }
gfCNCPoint3[6540] = {X 227.7203, Y 44.1697, Z -3.8333, A 0.000, B 0.000, C 0.000 }
gfCNCPoint3[6541] = {X 227.7205, Y 45.0000, Z -3.8333, A 0.000, B 0.000, C 0.000 }
gfCNCPoint3[6542] = {X 227.6142, Y 45.9435, Z -3.8333, A 0.000, B 0.000, C 0.000 }
gfCNCPoint3[6543] = {X 227.3006, Y 46.8397, Z -3.8333, A 0.000, B 0.000, C 0.000 }
gfCNCPoint3[6544] = {X 226.7954, Y 47.6436, Z -3.8333, A 0.000, B 0.000, C 0.000 }
gfCNCPoint3[6545] = {X 226.1241, Y 48.3150, Z -3.8333, A 0.000, B 0.000, C 0.000 }
gfCNCPoint3[6546] = {X 225.3201, Y 48.8201, Z -3.8333, A 0.000, B 0.000, C 0.000 }
gfCNCPoint3[6547] = {X 224.4240, Y 49.1337, Z -3.8333, A 0.000, B 0.000, C 0.000 }
gfCNCPoint3[6548] = {X 223.4805, Y 49.2400, Z -3.8333, A 0.000, B 0.000, C 0.000 }
gfCNCPoint3[6549] = {X 217.0370, Y 49.2400, Z -3.8333, A 0.000, B 0.000, C 0.000 }
gfCNCPoint3[6550] = {X 216.0982, Y 49.1348, Z -3.8333, A 0.000, B 0.000, C 0.000 }
gfCNCPoint3[6551] = {X 215.2061, Y 48.8243, Z -3.8333, A 0.000, B 0.000, C 0.000 }
gfCNCPoint3[6552] = {X 214.4048, Y 48.3240, Z -3.8333, A 0.000, B 0.000, C 0.000 }
gfCNCPoint3[6553] = {X 213.7341, Y 47.6587, Z -3.8333, A 0.000, B 0.000, C 0.000 }
gfCNCPoint3[6554] = {X 213.2275, Y 46.8614, Z -3.8333, A 0.000, B 0.000, C 0.000 }
gfCNCPoint3[6555] = {X 212.9099, Y 45.9717, Z -3.8333, A 0.000, B 0.000, C 0.000 }
gfCNCPoint3[6556] = {X 212.7972, Y 45.0338, Z -3.8333, A 0.000, B 0.000, C 0.000 }
gfCNCPoint3[6557] = {X 212.7970, Y 44.1967, Z -3.8333, A 0.000, B 0.000, C 0.000 }
gfCNCPoint3[6558] = {X 212.8675, Y 43.4329, Z -3.8333, A 0.000, B 0.000, C 0.000 }
gfCNCPoint3[6559] = {X 213.0767, Y 42.6949, Z -3.8333, A 0.000, B 0.000, C 0.000 }
gfCNCPoint3[6560] = {X 213.4174, Y 42.0077, Z -3.8333, A 0.000, B 0.000, C 0.000 }
gfCNCPoint3[6561] = {X 213.8781, Y 41.3945, Z -3.8333, A 0.000, B 0.000, C 0.000 }
gfCNCPoint3[6562] = {X 214.3206, Y 40.9065, Z -3.8333, A 0.000, B 0.000, C 0.000 }
gfCNCPoint3[6563] = {X 214.3252, Y 40.3065, Z -3.8333, A 0.000, B 0.000, C 0.000 }
gfCNCPoint3[6564] = {X 214.3252, Y 28.5741, Z -3.8333, A 0.000, B 0.000, C 0.000 }
gfCNCPoint3[6565] = {X 210.3252, Y 28.5741, Z -3.8333, A 0.000, B 0.000, C 0.000 }
gfCNCPoint3[6566] = {X 214.4052, Y 28.5741, Z -3.8333, A 0.000, B 0.000, C 0.000 }
gfCNCPoint3[6567] = {X 214.4052, Y 17.4617, Z -3.8333, A 0.000, B 0.000, C 0.000 }
gfCNCPoint3[6568] = {X 214.3999, Y 16.7692, Z -3.8333, A 0.000, B 0.000, C 0.000 }
gfCNCPoint3[6569] = {X 214.4034, Y 16.1982, Z -3.8333, A 0.000, B 0.000, C 0.000 }
gfCNCPoint3[6570] = {X 213.7661, Y 15.5484, Z -3.8333, A 0.000, B 0.000, C 0.000 }
gfCNCPoint3[6571] = {X 213.2854, Y 14.7756, Z -3.8333, A 0.000, B 0.000, C 0.000 }
gfCNCPoint3[6572] = {X 212.9843, Y 13.9167, Z -3.8333, A 0.000, B 0.000, C 0.000 }
gfCNCPoint3[6573] = {X 212.8772, Y 13.0130, Z -3.8333, A 0.000, B 0.000, C 0.000 }
gfCNCPoint3[6574] = {X 212.8770, Y 12.1868, Z -3.8333, A 0.000, B 0.000, C 0.000 }
gfCNCPoint3[6575] = {X 212.9813, Y 11.2611, Z -3.8333, A 0.000, B 0.000, C 0.000 }
gfCNCPoint3[6576] = {X 213.2890, Y 10.3819, Z -3.8333, A 0.000, B 0.000, C 0.000 }
gfCNCPoint3[6577] = {X 213.7846, Y 9.5931, Z -3.8333, A 0.000, B 0.000, C 0.000 }
gfCNCPoint3[6578] = {X 214.4433, Y 8.9344, Z -3.8333, A 0.000, B 0.000, C 0.000 }
gfCNCPoint3[6579] = {X 215.2321, Y 8.4388, Z -3.8333, A 0.000, B 0.000, C 0.000 }
gfCNCPoint3[6580] = {X 216.1113, Y 8.1311, Z -3.8333, A 0.000, B 0.000, C 0.000 }
gfCNCPoint3[6581] = {X 217.0370, Y 8.0268, Z -3.8333, A 0.000, B 0.000, C 0.000 }
gfCNCPoint3[6582] = {X 223.4805, Y 8.0268, Z -3.8333, A 0.000, B 0.000, C 0.000 }
gfCNCPoint3[6583] = {X 224.4062, Y 8.1311, Z -3.8333, A 0.000, B 0.000, C 0.000 }
gfCNCPoint3[6584] = {X 225.2854, Y 8.4388, Z -3.8333, A 0.000, B 0.000, C 0.000 }
gfCNCPoint3[6585] = {X 226.0742, Y 8.9344, Z -3.8333, A 0.000, B 0.000, C 0.000 }
gfCNCPoint3[6586] = {X 226.7329, Y 9.5931, Z -3.8333, A 0.000, B 0.000, C 0.000 }
gfCNCPoint3[6587] = {X 227.2285, Y 10.3819, Z -3.8333, A 0.000, B 0.000, C 0.000 }
gfCNCPoint3[6588] = {X 227.5362, Y 11.2611, Z -3.8333, A 0.000, B 0.000, C 0.000 }
gfCNCPoint3[6589] = {X 227.6405, Y 12.1868, Z -3.8333, A 0.000, B 0.000, C 0.000 }
gfCNCPoint3[6590] = {X 227.6405, Y 12.9781, Z -3.8333, A 0.000, B 0.000, C 0.000 }
gfCNCPoint3[6591] = {X 227.5389, Y 13.8917, Z -3.8333, A 0.000, B 0.000, C 0.000 }
gfCNCPoint3[6592] = {X 227.2392, Y 14.7606, Z -3.8333, A 0.000, B 0.000, C 0.000 }
gfCNCPoint3[6593] = {X 226.7560, Y 15.5425, Z -3.8333, A 0.000, B 0.000, C 0.000 }
gfCNCPoint3[6594] = {X 226.1129, Y 16.1992, Z -3.8333, A 0.000, B 0.000, C 0.000 }
gfCNCPoint3[6595] = {X 226.1139, Y 40.9904, Z -3.8333, A 0.000, B 0.000, C 0.000 }
gfCNCPoint3[6596] = {X 226.7504, Y 41.6391, Z -3.8333, A 0.000, B 0.000, C 0.000 }
gfCNCPoint3[6597] = {X 227.2308, Y 42.4106, Z -3.8333, A 0.000, B 0.000, C 0.000 }
gfCNCPoint3[6598] = {X 227.5323, Y 43.2680, Z -3.8333, A 0.000, B 0.000, C 0.000 }
gfCNCPoint3[6599] = {X 227.6403, Y 44.1704, Z -3.8333, A 0.000, B 0.000, C 0.000 }
gfCNCPoint3[6600] = {X 227.6405, Y 45.0000, Z -3.8333, A 0.000, B 0.000, C 0.000 }
gfCNCPoint3[6601] = {X 227.5362, Y 45.9257, Z -3.8333, A 0.000, B 0.000, C 0.000 }
gfCNCPoint3[6602] = {X 227.2285, Y 46.8050, Z -3.8333, A 0.000, B 0.000, C 0.000 }
gfCNCPoint3[6603] = {X 226.7329, Y 47.5937, Z -3.8333, A 0.000, B 0.000, C 0.000 }
gfCNCPoint3[6604] = {X 226.0742, Y 48.2524, Z -3.8333, A 0.000, B 0.000, C 0.000 }
gfCNCPoint3[6605] = {X 225.2854, Y 48.7480, Z -3.8333, A 0.000, B 0.000, C 0.000 }
gfCNCPoint3[6606] = {X 224.4062, Y 49.0557, Z -3.8333, A 0.000, B 0.000, C 0.000 }
gfCNCPoint3[6607] = {X 223.4805, Y 49.1600, Z -3.8333, A 0.000, B 0.000, C 0.000 }
gfCNCPoint3[6608] = {X 217.0370, Y 49.1600, Z -3.8333, A 0.000, B 0.000, C 0.000 }
gfCNCPoint3[6609] = {X 216.1160, Y 49.0568, Z -3.8333, A 0.000, B 0.000, C 0.000 }
gfCNCPoint3[6610] = {X 215.2406, Y 48.7521, Z -3.8333, A 0.000, B 0.000, C 0.000 }
gfCNCPoint3[6611] = {X 214.4544, Y 48.2613, Z -3.8333, A 0.000, B 0.000, C 0.000 }
gfCNCPoint3[6612] = {X 213.7965, Y 47.6085, Z -3.8333, A 0.000, B 0.000, C 0.000 }
gfCNCPoint3[6613] = {X 213.2993, Y 46.8263, Z -3.8333, A 0.000, B 0.000, C 0.000 }
gfCNCPoint3[6614] = {X 212.9877, Y 45.9534, Z -3.8333, A 0.000, B 0.000, C 0.000 }
gfCNCPoint3[6615] = {X 212.8771, Y 45.0332, Z -3.8333, A 0.000, B 0.000, C 0.000 }
gfCNCPoint3[6616] = {X 212.8770, Y 44.1967, Z -3.8333, A 0.000, B 0.000, C 0.000 }
gfCNCPoint3[6617] = {X 212.9462, Y 43.4475, Z -3.8333, A 0.000, B 0.000, C 0.000 }
gfCNCPoint3[6618] = {X 213.1513, Y 42.7237, Z -3.8333, A 0.000, B 0.000, C 0.000 }
gfCNCPoint3[6619] = {X 213.4855, Y 42.0497, Z -3.8333, A 0.000, B 0.000, C 0.000 }
gfCNCPoint3[6620] = {X 213.9374, Y 41.4483, Z -3.8333, A 0.000, B 0.000, C 0.000 }
gfCNCPoint3[6621] = {X 214.4004, Y 40.9376, Z -3.8333, A 0.000, B 0.000, C 0.000 }
gfCNCPoint3[6622] = {X 214.4052, Y 40.3069, Z -3.8333, A 0.000, B 0.000, C 0.000 }
gfCNCPoint3[6623] = {X 214.4052, Y 28.5741, Z -3.8333, A 0.000, B 0.000, C 0.000 }
gfCNCPoint3[6624] = {X 210.4052, Y 28.5741, Z -3.8333, A 0.000, B 0.000, C 0.000 }
gfCNCPoint3[6625] = {X 214.4852, Y 28.5741, Z -3.8333, A 0.000, B 0.000, C 0.000 }
gfCNCPoint3[6626] = {X 214.4852, Y 17.4614, Z -3.8333, A 0.000, B 0.000, C 0.000 }
gfCNCPoint3[6627] = {X 214.4799, Y 16.7691, Z -3.8333, A 0.000, B 0.000, C 0.000 }
gfCNCPoint3[6628] = {X 214.4836, Y 16.1602, Z -3.8333, A 0.000, B 0.000, C 0.000 }
gfCNCPoint3[6629] = {X 214.4257, Y 16.1129, Z -3.8333, A 0.000, B 0.000, C 0.000 }
gfCNCPoint3[6630] = {X 214.3687, Y 16.0645, Z -3.8333, A 0.000, B 0.000, C 0.000 }
gfCNCPoint3[6631] = {X 213.7780, Y 15.4327, Z -3.8333, A 0.000, B 0.000, C 0.000 }
gfCNCPoint3[6632] = {X 213.3338, Y 14.6906, Z -3.8333, A 0.000, B 0.000, C 0.000 }
gfCNCPoint3[6633] = {X 213.0561, Y 13.8715, Z -3.8333, A 0.000, B 0.000, C 0.000 }
gfCNCPoint3[6634] = {X 212.9572, Y 13.0123, Z -3.8333, A 0.000, B 0.000, C 0.000 }
gfCNCPoint3[6635] = {X 212.9570, Y 12.1868, Z -3.8333, A 0.000, B 0.000, C 0.000 }
gfCNCPoint3[6636] = {X 213.0593, Y 11.2789, Z -3.8333, A 0.000, B 0.000, C 0.000 }
gfCNCPoint3[6637] = {X 213.3611, Y 10.4166, Z -3.8333, A 0.000, B 0.000, C 0.000 }
gfCNCPoint3[6638] = {X 213.8471, Y 9.6430, Z -3.8333, A 0.000, B 0.000, C 0.000 }
gfCNCPoint3[6639] = {X 214.4932, Y 8.9969, Z -3.8333, A 0.000, B 0.000, C 0.000 }
gfCNCPoint3[6640] = {X 215.2668, Y 8.5109, Z -3.8333, A 0.000, B 0.000, C 0.000 }
gfCNCPoint3[6641] = {X 216.1291, Y 8.2091, Z -3.8333, A 0.000, B 0.000, C 0.000 }
gfCNCPoint3[6642] = {X 217.0370, Y 8.1068, Z -3.8333, A 0.000, B 0.000, C 0.000 }
gfCNCPoint3[6643] = {X 223.4805, Y 8.1068, Z -3.8333, A 0.000, B 0.000, C 0.000 }
gfCNCPoint3[6644] = {X 224.3884, Y 8.2091, Z -3.8333, A 0.000, B 0.000, C 0.000 }
gfCNCPoint3[6645] = {X 225.2507, Y 8.5109, Z -3.8333, A 0.000, B 0.000, C 0.000 }
gfCNCPoint3[6646] = {X 226.0243, Y 8.9969, Z -3.8333, A 0.000, B 0.000, C 0.000 }
gfCNCPoint3[6647] = {X 226.6704, Y 9.6430, Z -3.8333, A 0.000, B 0.000, C 0.000 }
gfCNCPoint3[6648] = {X 227.1564, Y 10.4166, Z -3.8333, A 0.000, B 0.000, C 0.000 }
gfCNCPoint3[6649] = {X 227.4582, Y 11.2789, Z -3.8333, A 0.000, B 0.000, C 0.000 }
gfCNCPoint3[6650] = {X 227.5605, Y 12.1868, Z -3.8333, A 0.000, B 0.000, C 0.000 }
gfCNCPoint3[6651] = {X 227.5605, Y 12.9781, Z -3.8333, A 0.000, B 0.000, C 0.000 }
gfCNCPoint3[6652] = {X 227.4588, Y 13.8833, Z -3.8333, A 0.000, B 0.000, C 0.000 }
gfCNCPoint3[6653] = {X 227.1588, Y 14.7433, Z -3.8333, A 0.000, B 0.000, C 0.000 }
gfCNCPoint3[6654] = {X 226.6755, Y 15.5154, Z -3.8333, A 0.000, B 0.000, C 0.000 }
gfCNCPoint3[6655] = {X 226.0329, Y 16.1610, Z -3.8333, A 0.000, B 0.000, C 0.000 }
gfCNCPoint3[6656] = {X 226.0339, Y 41.0285, Z -3.8333, A 0.000, B 0.000, C 0.000 }
gfCNCPoint3[6657] = {X 226.1410, Y 41.1155, Z -3.8333, A 0.000, B 0.000, C 0.000 }
gfCNCPoint3[6658] = {X 226.7343, Y 41.7472, Z -3.8333, A 0.000, B 0.000, C 0.000 }
gfCNCPoint3[6659] = {X 227.1808, Y 42.4900, Z -3.8333, A 0.000, B 0.000, C 0.000 }
gfCNCPoint3[6660] = {X 227.4603, Y 43.3103, Z -3.8333, A 0.000, B 0.000, C 0.000 }
gfCNCPoint3[6661] = {X 227.5603, Y 44.1712, Z -3.8333, A 0.000, B 0.000, C 0.000 }
gfCNCPoint3[6662] = {X 227.5605, Y 45.0000, Z -3.8333, A 0.000, B 0.000, C 0.000 }
gfCNCPoint3[6663] = {X 227.4582, Y 45.9079, Z -3.8333, A 0.000, B 0.000, C 0.000 }
gfCNCPoint3[6664] = {X 227.1564, Y 46.7702, Z -3.8333, A 0.000, B 0.000, C 0.000 }
gfCNCPoint3[6665] = {X 226.6704, Y 47.5438, Z -3.8333, A 0.000, B 0.000, C 0.000 }
gfCNCPoint3[6666] = {X 226.0243, Y 48.1899, Z -3.8333, A 0.000, B 0.000, C 0.000 }
gfCNCPoint3[6667] = {X 225.2507, Y 48.6760, Z -3.8333, A 0.000, B 0.000, C 0.000 }
gfCNCPoint3[6668] = {X 224.3884, Y 48.9777, Z -3.8333, A 0.000, B 0.000, C 0.000 }
gfCNCPoint3[6669] = {X 223.4805, Y 49.0800, Z -3.8333, A 0.000, B 0.000, C 0.000 }
gfCNCPoint3[6670] = {X 217.0370, Y 49.0800, Z -3.8333, A 0.000, B 0.000, C 0.000 }
gfCNCPoint3[6671] = {X 216.1337, Y 48.9787, Z -3.8333, A 0.000, B 0.000, C 0.000 }
gfCNCPoint3[6672] = {X 215.2752, Y 48.6800, Z -3.8333, A 0.000, B 0.000, C 0.000 }
gfCNCPoint3[6673] = {X 214.5041, Y 48.1986, Z -3.8333, A 0.000, B 0.000, C 0.000 }
gfCNCPoint3[6674] = {X 213.8588, Y 47.5584, Z -3.8333, A 0.000, B 0.000, C 0.000 }
gfCNCPoint3[6675] = {X 213.3712, Y 46.7912, Z -3.8333, A 0.000, B 0.000, C 0.000 }
gfCNCPoint3[6676] = {X 213.0656, Y 45.9351, Z -3.8333, A 0.000, B 0.000, C 0.000 }
gfCNCPoint3[6677] = {X 212.9571, Y 45.0325, Z -3.8333, A 0.000, B 0.000, C 0.000 }
gfCNCPoint3[6678] = {X 212.9570, Y 44.1967, Z -3.8333, A 0.000, B 0.000, C 0.000 }
gfCNCPoint3[6679] = {X 213.0248, Y 43.4622, Z -3.8333, A 0.000, B 0.000, C 0.000 }
gfCNCPoint3[6680] = {X 213.2259, Y 42.7525, Z -3.8333, A 0.000, B 0.000, C 0.000 }
gfCNCPoint3[6681] = {X 213.5536, Y 42.0917, Z -3.8333, A 0.000, B 0.000, C 0.000 }
gfCNCPoint3[6682] = {X 213.9967, Y 41.5020, Z -3.8333, A 0.000, B 0.000, C 0.000 }
gfCNCPoint3[6683] = {X 214.4801, Y 40.9687, Z -3.8333, A 0.000, B 0.000, C 0.000 }
gfCNCPoint3[6684] = {X 214.4852, Y 40.3072, Z -3.8333, A 0.000, B 0.000, C 0.000 }
gfCNCPoint3[6685] = {X 214.4852, Y 28.5741, Z -3.8333, A 0.000, B 0.000, C 0.000 }
gfCNCPoint3[6686] = {X 210.4852, Y 28.5741, Z -3.8333, A 0.000, B 0.000, C 0.000 }
gfCNCPoint3[6687] = {X 214.5652, Y 28.5741, Z -3.8333, A 0.000, B 0.000, C 0.000 }
gfCNCPoint3[6688] = {X 214.5652, Y 17.4611, Z -3.8333, A 0.000, B 0.000, C 0.000 }
gfCNCPoint3[6689] = {X 214.5599, Y 16.7687, Z -3.8333, A 0.000, B 0.000, C 0.000 }
gfCNCPoint3[6690] = {X 214.5592, Y 16.1865, Z -3.8333, A 0.000, B 0.000, C 0.000 }
gfCNCPoint3[6691] = {X 214.5756, Y 16.1310, Z -3.8333, A 0.000, B 0.000, C 0.000 }
gfCNCPoint3[6692] = {X 214.4975, Y 16.0685, Z -3.8333, A 0.000, B 0.000, C 0.000 }
gfCNCPoint3[6693] = {X 214.4210, Y 16.0040, Z -3.8333, A 0.000, B 0.000, C 0.000 }
gfCNCPoint3[6694] = {X 213.8369, Y 15.3778, Z -3.8333, A 0.000, B 0.000, C 0.000 }
gfCNCPoint3[6695] = {X 213.3994, Y 14.6417, Z -3.8333, A 0.000, B 0.000, C 0.000 }
gfCNCPoint3[6696] = {X 213.1287, Y 13.8293, Z -3.8333, A 0.000, B 0.000, C 0.000 }
gfCNCPoint3[6697] = {X 213.0370, Y 12.9779, Z -3.8333, A 0.000, B 0.000, C 0.000 }
gfCNCPoint3[6698] = {X 213.0370, Y 12.1868, Z -3.8333, A 0.000, B 0.000, C 0.000 }
gfCNCPoint3[6699] = {X 213.1373, Y 11.2967, Z -3.8333, A 0.000, B 0.000, C 0.000 }
gfCNCPoint3[6700] = {X 213.4331, Y 10.4513, Z -3.8333, A 0.000, B 0.000, C 0.000 }
gfCNCPoint3[6701] = {X 213.9097, Y 9.6929, Z -3.8333, A 0.000, B 0.000, C 0.000 }
gfCNCPoint3[6702] = {X 214.5431, Y 9.0595, Z -3.8333, A 0.000, B 0.000, C 0.000 }
gfCNCPoint3[6703] = {X 215.3015, Y 8.5829, Z -3.8333, A 0.000, B 0.000, C 0.000 }
gfCNCPoint3[6704] = {X 216.1469, Y 8.2871, Z -3.8333, A 0.000, B 0.000, C 0.000 }
gfCNCPoint3[6705] = {X 217.0370, Y 8.1868, Z -3.8333, A 0.000, B 0.000, C 0.000 }
gfCNCPoint3[6706] = {X 223.4805, Y 8.1868, Z -3.8333, A 0.000, B 0.000, C 0.000 }
gfCNCPoint3[6707] = {X 224.3706, Y 8.2871, Z -3.8333, A 0.000, B 0.000, C 0.000 }
gfCNCPoint3[6708] = {X 225.2160, Y 8.5829, Z -3.8333, A 0.000, B 0.000, C 0.000 }
gfCNCPoint3[6709] = {X 225.9744, Y 9.0595, Z -3.8333, A 0.000, B 0.000, C 0.000 }
gfCNCPoint3[6710] = {X 226.6078, Y 9.6929, Z -3.8333, A 0.000, B 0.000, C 0.000 }
gfCNCPoint3[6711] = {X 227.0844, Y 10.4513, Z -3.8333, A 0.000, B 0.000, C 0.000 }
gfCNCPoint3[6712] = {X 227.3802, Y 11.2967, Z -3.8333, A 0.000, B 0.000, C 0.000 }
gfCNCPoint3[6713] = {X 227.4805, Y 12.1868, Z -3.8333, A 0.000, B 0.000, C 0.000 }
gfCNCPoint3[6714] = {X 227.4803, Y 13.0192, Z -3.8333, A 0.000, B 0.000, C 0.000 }
gfCNCPoint3[6715] = {X 227.3716, Y 13.9049, Z -3.8333, A 0.000, B 0.000, C 0.000 }
gfCNCPoint3[6716] = {X 227.0693, Y 14.7444, Z -3.8333, A 0.000, B 0.000, C 0.000 }
gfCNCPoint3[6717] = {X 226.5885, Y 15.4960, Z -3.8333, A 0.000, B 0.000, C 0.000 }
gfCNCPoint3[6718] = {X 225.9529, Y 16.1224, Z -3.8333, A 0.000, B 0.000, C 0.000 }
gfCNCPoint3[6719] = {X 225.9539, Y 41.0665, Z -3.8333, A 0.000, B 0.000, C 0.000 }
gfCNCPoint3[6720] = {X 226.0926, Y 41.1795, Z -3.8333, A 0.000, B 0.000, C 0.000 }
gfCNCPoint3[6721] = {X 226.6783, Y 41.8059, Z -3.8333, A 0.000, B 0.000, C 0.000 }
gfCNCPoint3[6722] = {X 227.1170, Y 42.5428, Z -3.8333, A 0.000, B 0.000, C 0.000 }
gfCNCPoint3[6723] = {X 227.3886, Y 43.3563, Z -3.8333, A 0.000, B 0.000, C 0.000 }
gfCNCPoint3[6724] = {X 227.4805, Y 44.2089, Z -3.8333, A 0.000, B 0.000, C 0.000 }
gfCNCPoint3[6725] = {X 227.4805, Y 45.0000, Z -3.8333, A 0.000, B 0.000, C 0.000 }
gfCNCPoint3[6726] = {X 227.3802, Y 45.8901, Z -3.8333, A 0.000, B 0.000, C 0.000 }
gfCNCPoint3[6727] = {X 227.0844, Y 46.7355, Z -3.8333, A 0.000, B 0.000, C 0.000 }
gfCNCPoint3[6728] = {X 226.6078, Y 47.4940, Z -3.8333, A 0.000, B 0.000, C 0.000 }
gfCNCPoint3[6729] = {X 225.9744, Y 48.1273, Z -3.8333, A 0.000, B 0.000, C 0.000 }
gfCNCPoint3[6730] = {X 225.2160, Y 48.6039, Z -3.8333, A 0.000, B 0.000, C 0.000 }
gfCNCPoint3[6731] = {X 224.3706, Y 48.8997, Z -3.8333, A 0.000, B 0.000, C 0.000 }
gfCNCPoint3[6732] = {X 223.4805, Y 49.0000, Z -3.8333, A 0.000, B 0.000, C 0.000 }
gfCNCPoint3[6733] = {X 217.0370, Y 49.0000, Z -3.8333, A 0.000, B 0.000, C 0.000 }
gfCNCPoint3[6734] = {X 216.1469, Y 48.8997, Z -3.8333, A 0.000, B 0.000, C 0.000 }
gfCNCPoint3[6735] = {X 215.3015, Y 48.6039, Z -3.8333, A 0.000, B 0.000, C 0.000 }
gfCNCPoint3[6736] = {X 214.5430, Y 48.1273, Z -3.8333, A 0.000, B 0.000, C 0.000 }
gfCNCPoint3[6737] = {X 213.9097, Y 47.4939, Z -3.8333, A 0.000, B 0.000, C 0.000 }
gfCNCPoint3[6738] = {X 213.4331, Y 46.7355, Z -3.8333, A 0.000, B 0.000, C 0.000 }
gfCNCPoint3[6739] = {X 213.1373, Y 45.8901, Z -3.8333, A 0.000, B 0.000, C 0.000 }
gfCNCPoint3[6740] = {X 213.0370, Y 45.0000, Z -3.8333, A 0.000, B 0.000, C 0.000 }
gfCNCPoint3[6741] = {X 213.0370, Y 44.1967, Z -3.8333, A 0.000, B 0.000, C 0.000 }
gfCNCPoint3[6742] = {X 213.1549, Y 43.2411, Z -3.8333, A 0.000, B 0.000, C 0.000 }
gfCNCPoint3[6743] = {X 213.5015, Y 42.3428, Z -3.8333, A 0.000, B 0.000, C 0.000 }
gfCNCPoint3[6744] = {X 214.0559, Y 41.5557, Z -3.8333, A 0.000, B 0.000, C 0.000 }
gfCNCPoint3[6745] = {X 214.5599, Y 40.9999, Z -3.8333, A 0.000, B 0.000, C 0.000 }
gfCNCPoint3[6746] = {X 214.5652, Y 40.3075, Z -3.8333, A 0.000, B 0.000, C 0.000 }
gfCNCPoint3[6747] = {X 214.5652, Y 28.5741, Z -3.8333, A 0.000, B 0.000, C 0.000 }
gfCNCPoint3[6748] = {X 210.4852, Y 28.5741, Z -3.8333, A 0.000, B 0.000, C 0.000 }
gfCNCPoint3[6749] = {X 210.4852, Y 28.5741, Z -0.8333, A 0.000, B 0.000, C 0.000 }
gfCNCPoint3[6750] = {X 210.4852, Y 28.5741, Z 11.0000, A 0.000, B 0.000, C 0.000 }
gfCNCPoint3[6751] = {X 273.6036, Y 28.5936, Z 11.0000, A 0.000, B 0.000, C 0.000 }
gfCNCPoint3[6752] = {X 273.6036, Y 28.5936, Z -0.8333, A 0.000, B 0.000, C 0.000 }
gfCNCPoint3[6753] = {X 273.6036, Y 28.5936, Z -3.8333, A 0.000, B 0.000, C 0.000 }
gfCNCPoint3[6754] = {X 269.5236, Y 28.5936, Z -3.8333, A 0.000, B 0.000, C 0.000 }
gfCNCPoint3[6755] = {X 269.5235, Y 40.9133, Z -3.8333, A 0.000, B 0.000, C 0.000 }
gfCNCPoint3[6756] = {X 269.5372, Y 40.9243, Z -3.8333, A 0.000, B 0.000, C 0.000 }
gfCNCPoint3[6757] = {X 270.1697, Y 41.5939, Z -3.8333, A 0.000, B 0.000, C 0.000 }
gfCNCPoint3[6758] = {X 270.6459, Y 42.3823, Z -3.8333, A 0.000, B 0.000, C 0.000 }
gfCNCPoint3[6759] = {X 270.9441, Y 43.2537, Z -3.8333, A 0.000, B 0.000, C 0.000 }
gfCNCPoint3[6760] = {X 271.0508, Y 44.1686, Z -3.8333, A 0.000, B 0.000, C 0.000 }
gfCNCPoint3[6761] = {X 271.0510, Y 45.0000, Z -3.8333, A 0.000, B 0.000, C 0.000 }
gfCNCPoint3[6762] = {X 270.9427, Y 45.9613, Z -3.8333, A 0.000, B 0.000, C 0.000 }
gfCNCPoint3[6763] = {X 270.6232, Y 46.8744, Z -3.8333, A 0.000, B 0.000, C 0.000 }
gfCNCPoint3[6764] = {X 270.1085, Y 47.6935, Z -3.8333, A 0.000, B 0.000, C 0.000 }
gfCNCPoint3[6765] = {X 269.4245, Y 48.3775, Z -3.8333, A 0.000, B 0.000, C 0.000 }
gfCNCPoint3[6766] = {X 268.6054, Y 48.8922, Z -3.8333, A 0.000, B 0.000, C 0.000 }
gfCNCPoint3[6767] = {X 267.6923, Y 49.2117, Z -3.8333, A 0.000, B 0.000, C 0.000 }
gfCNCPoint3[6768] = {X 266.7310, Y 49.3200, Z -3.8333, A 0.000, B 0.000, C 0.000 }
gfCNCPoint3[6769] = {X 260.2876, Y 49.3200, Z -3.8333, A 0.000, B 0.000, C 0.000 }
gfCNCPoint3[6770] = {X 259.3310, Y 49.2128, Z -3.8333, A 0.000, B 0.000, C 0.000 }
gfCNCPoint3[6771] = {X 258.4219, Y 48.8963, Z -3.8333, A 0.000, B 0.000, C 0.000 }
gfCNCPoint3[6772] = {X 257.6054, Y 48.3865, Z -3.8333, A 0.000, B 0.000, C 0.000 }
gfCNCPoint3[6773] = {X 256.9221, Y 47.7085, Z -3.8333, A 0.000, B 0.000, C 0.000 }
gfCNCPoint3[6774] = {X 256.4059, Y 46.8960, Z -3.8333, A 0.000, B 0.000, C 0.000 }
gfCNCPoint3[6775] = {X 256.0824, Y 45.9894, Z -3.8333, A 0.000, B 0.000, C 0.000 }
gfCNCPoint3[6776] = {X 255.9677, Y 45.0336, Z -3.8333, A 0.000, B 0.000, C 0.000 }
gfCNCPoint3[6777] = {X 255.9680, Y 44.1494, Z -3.8333, A 0.000, B 0.000, C 0.000 }
gfCNCPoint3[6778] = {X 256.0784, Y 43.2364, Z -3.8333, A 0.000, B 0.000, C 0.000 }
gfCNCPoint3[6779] = {X 256.3796, Y 42.3675, Z -3.8333, A 0.000, B 0.000, C 0.000 }
gfCNCPoint3[6780] = {X 256.8579, Y 41.5821, Z -3.8333, A 0.000, B 0.000, C 0.000 }
gfCNCPoint3[6781] = {X 257.4915, Y 40.9157, Z -3.8333, A 0.000, B 0.000, C 0.000 }
gfCNCPoint3[6782] = {X 257.4915, Y 34.4738, Z -3.8333, A 0.000, B 0.000, C 0.000 }
gfCNCPoint3[6783] = {X 254.7674, Y 34.4738, Z -3.8333, A 0.000, B 0.000, C 0.000 }
gfCNCPoint3[6784] = {X 250.4837, Y 42.8184, Z -3.8333, A 0.000, B 0.000, C 0.000 }
gfCNCPoint3[6785] = {X 250.6527, Y 43.4862, Z -3.8333, A 0.000, B 0.000, C 0.000 }
gfCNCPoint3[6786] = {X 250.7134, Y 44.1723, Z -3.8333, A 0.000, B 0.000, C 0.000 }
gfCNCPoint3[6787] = {X 250.7136, Y 45.0000, Z -3.8333, A 0.000, B 0.000, C 0.000 }
gfCNCPoint3[6788] = {X 250.6052, Y 45.9613, Z -3.8333, A 0.000, B 0.000, C 0.000 }
gfCNCPoint3[6789] = {X 250.2857, Y 46.8744, Z -3.8333, A 0.000, B 0.000, C 0.000 }
gfCNCPoint3[6790] = {X 249.7711, Y 47.6935, Z -3.8333, A 0.000, B 0.000, C 0.000 }
gfCNCPoint3[6791] = {X 249.0870, Y 48.3775, Z -3.8333, A 0.000, B 0.000, C 0.000 }
gfCNCPoint3[6792] = {X 248.2679, Y 48.8922, Z -3.8333, A 0.000, B 0.000, C 0.000 }
gfCNCPoint3[6793] = {X 247.3548, Y 49.2117, Z -3.8333, A 0.000, B 0.000, C 0.000 }
gfCNCPoint3[6794] = {X 246.3936, Y 49.3200, Z -3.8333, A 0.000, B 0.000, C 0.000 }
gfCNCPoint3[6795] = {X 239.8075, Y 49.3200, Z -3.8333, A 0.000, B 0.000, C 0.000 }
gfCNCPoint3[6796] = {X 238.8462, Y 49.2117, Z -3.8333, A 0.000, B 0.000, C 0.000 }
gfCNCPoint3[6797] = {X 237.9331, Y 48.8922, Z -3.8333, A 0.000, B 0.000, C 0.000 }
gfCNCPoint3[6798] = {X 237.1141, Y 48.3775, Z -3.8333, A 0.000, B 0.000, C 0.000 }
gfCNCPoint3[6799] = {X 236.4300, Y 47.6935, Z -3.8333, A 0.000, B 0.000, C 0.000 }
gfCNCPoint3[6800] = {X 235.9153, Y 46.8745, Z -3.8333, A 0.000, B 0.000, C 0.000 }
gfCNCPoint3[6801] = {X 235.5958, Y 45.9614, Z -3.8333, A 0.000, B 0.000, C 0.000 }
gfCNCPoint3[6802] = {X 235.4875, Y 45.0001, Z -3.8333, A 0.000, B 0.000, C 0.000 }
gfCNCPoint3[6803] = {X 235.4879, Y 44.1494, Z -3.8333, A 0.000, B 0.000, C 0.000 }
gfCNCPoint3[6804] = {X 235.5856, Y 43.2935, Z -3.8333, A 0.000, B 0.000, C 0.000 }
gfCNCPoint3[6805] = {X 235.8511, Y 42.4740, Z -3.8333, A 0.000, B 0.000, C 0.000 }
gfCNCPoint3[6806] = {X 236.2739, Y 41.7236, Z -3.8333, A 0.000, B 0.000, C 0.000 }
gfCNCPoint3[6807] = {X 236.8373, Y 41.0719, Z -3.8333, A 0.000, B 0.000, C 0.000 }
gfCNCPoint3[6808] = {X 237.5187, Y 40.5449, Z -3.8333, A 0.000, B 0.000, C 0.000 }
gfCNCPoint3[6809] = {X 238.2911, Y 40.1637, Z -3.8333, A 0.000, B 0.000, C 0.000 }
gfCNCPoint3[6810] = {X 242.2804, Y 32.3551, Z -3.8333, A 0.000, B 0.000, C 0.000 }
gfCNCPoint3[6811] = {X 241.1104, Y 31.5688, Z -3.8333, A 0.000, B 0.000, C 0.000 }
gfCNCPoint3[6812] = {X 240.0472, Y 30.6431, Z -3.8333, A 0.000, B 0.000, C 0.000 }
gfCNCPoint3[6813] = {X 239.1074, Y 29.5924, Z -3.8333, A 0.000, B 0.000, C 0.000 }
gfCNCPoint3[6814] = {X 238.3055, Y 28.4330, Z -3.8333, A 0.000, B 0.000, C 0.000 }
gfCNCPoint3[6815] = {X 237.6540, Y 27.1829, Z -3.8333, A 0.000, B 0.000, C 0.000 }
gfCNCPoint3[6816] = {X 237.1629, Y 25.8614, Z -3.8333, A 0.000, B 0.000, C 0.000 }
gfCNCPoint3[6817] = {X 236.7428, Y 24.0500, Z -3.8333, A 0.000, B 0.000, C 0.000 }
gfCNCPoint3[6818] = {X 236.5286, Y 22.2028, Z -3.8333, A 0.000, B 0.000, C 0.000 }
gfCNCPoint3[6819] = {X 236.5233, Y 20.3433, Z -3.8333, A 0.000, B 0.000, C 0.000 }
gfCNCPoint3[6820] = {X 236.7267, Y 18.4950, Z -3.8333, A 0.000, B 0.000, C 0.000 }
gfCNCPoint3[6821] = {X 237.1364, Y 16.6811, Z -3.8333, A 0.000, B 0.000, C 0.000 }
gfCNCPoint3[6822] = {X 237.7068, Y 15.1055, Z -3.8333, A 0.000, B 0.000, C 0.000 }
gfCNCPoint3[6823] = {X 238.4937, Y 13.6260, Z -3.8333, A 0.000, B 0.000, C 0.000 }
gfCNCPoint3[6824] = {X 239.4815, Y 12.2724, Z -3.8333, A 0.000, B 0.000, C 0.000 }
gfCNCPoint3[6825] = {X 240.6504, Y 11.0717, Z -3.8333, A 0.000, B 0.000, C 0.000 }
gfCNCPoint3[6826] = {X 241.9770, Y 10.0479, Z -3.8333, A 0.000, B 0.000, C 0.000 }
gfCNCPoint3[6827] = {X 243.4348, Y 9.2216, Z -3.8333, A 0.000, B 0.000, C 0.000 }
gfCNCPoint3[6828] = {X 244.9946, Y 8.6091, Z -3.8333, A 0.000, B 0.000, C 0.000 }
gfCNCPoint3[6829] = {X 246.6252, Y 8.2229, Z -3.8333, A 0.000, B 0.000, C 0.000 }
gfCNCPoint3[6830] = {X 248.7221, Y 7.9515, Z -3.8333, A 0.000, B 0.000, C 0.000 }
gfCNCPoint3[6831] = {X 250.8349, Y 7.8709, Z -3.8333, A 0.000, B 0.000, C 0.000 }
gfCNCPoint3[6832] = {X 266.7634, Y 7.8709, Z -3.8333, A 0.000, B 0.000, C 0.000 }
gfCNCPoint3[6833] = {X 267.7185, Y 7.9857, Z -3.8333, A 0.000, B 0.000, C 0.000 }
gfCNCPoint3[6834] = {X 268.6246, Y 8.3088, Z -3.8333, A 0.000, B 0.000, C 0.000 }
gfCNCPoint3[6835] = {X 269.4368, Y 8.8244, Z -3.8333, A 0.000, B 0.000, C 0.000 }
gfCNCPoint3[6836] = {X 270.1148, Y 9.5068, Z -3.8333, A 0.000, B 0.000, C 0.000 }
gfCNCPoint3[6837] = {X 270.6251, Y 10.3223, Z -3.8333, A 0.000, B 0.000, C 0.000 }
gfCNCPoint3[6838] = {X 270.9424, Y 11.2305, Z -3.8333, A 0.000, B 0.000, C 0.000 }
gfCNCPoint3[6839] = {X 271.0510, Y 12.1864, Z -3.8333, A 0.000, B 0.000, C 0.000 }
gfCNCPoint3[6840] = {X 271.0508, Y 13.0225, Z -3.8333, A 0.000, B 0.000, C 0.000 }
gfCNCPoint3[6841] = {X 270.9424, Y 13.9405, Z -3.8333, A 0.000, B 0.000, C 0.000 }
gfCNCPoint3[6842] = {X 270.6413, Y 14.8145, Z -3.8333, A 0.000, B 0.000, C 0.000 }
gfCNCPoint3[6843] = {X 270.1610, Y 15.6043, Z -3.8333, A 0.000, B 0.000, C 0.000 }
gfCNCPoint3[6844] = {X 269.5237, Y 16.2740, Z -3.8333, A 0.000, B 0.000, C 0.000 }
gfCNCPoint3[6845] = {X 269.5236, Y 28.5936, Z -3.8333, A 0.000, B 0.000, C 0.000 }
gfCNCPoint3[6846] = {X 273.5236, Y 28.5936, Z -3.8333, A 0.000, B 0.000, C 0.000 }
gfCNCPoint3[6847] = {X 269.4436, Y 28.5936, Z -3.8333, A 0.000, B 0.000, C 0.000 }
gfCNCPoint3[6848] = {X 269.4435, Y 40.9514, Z -3.8333, A 0.000, B 0.000, C 0.000 }
gfCNCPoint3[6849] = {X 269.4861, Y 40.9858, Z -3.8333, A 0.000, B 0.000, C 0.000 }
gfCNCPoint3[6850] = {X 270.1065, Y 41.6429, Z -3.8333, A 0.000, B 0.000, C 0.000 }
gfCNCPoint3[6851] = {X 270.5736, Y 42.4166, Z -3.8333, A 0.000, B 0.000, C 0.000 }
gfCNCPoint3[6852] = {X 270.8662, Y 43.2717, Z -3.8333, A 0.000, B 0.000, C 0.000 }
gfCNCPoint3[6853] = {X 270.9708, Y 44.1693, Z -3.8333, A 0.000, B 0.000, C 0.000 }
gfCNCPoint3[6854] = {X 270.9710, Y 45.0000, Z -3.8333, A 0.000, B 0.000, C 0.000 }
gfCNCPoint3[6855] = {X 270.8647, Y 45.9435, Z -3.8333, A 0.000, B 0.000, C 0.000 }
gfCNCPoint3[6856] = {X 270.5511, Y 46.8397, Z -3.8333, A 0.000, B 0.000, C 0.000 }
gfCNCPoint3[6857] = {X 270.0460, Y 47.6436, Z -3.8333, A 0.000, B 0.000, C 0.000 }
gfCNCPoint3[6858] = {X 269.3746, Y 48.3150, Z -3.8333, A 0.000, B 0.000, C 0.000 }
gfCNCPoint3[6859] = {X 268.5707, Y 48.8201, Z -3.8333, A 0.000, B 0.000, C 0.000 }
gfCNCPoint3[6860] = {X 267.6745, Y 49.1337, Z -3.8333, A 0.000, B 0.000, C 0.000 }
gfCNCPoint3[6861] = {X 266.7310, Y 49.2400, Z -3.8333, A 0.000, B 0.000, C 0.000 }
gfCNCPoint3[6862] = {X 260.2876, Y 49.2400, Z -3.8333, A 0.000, B 0.000, C 0.000 }
gfCNCPoint3[6863] = {X 259.3487, Y 49.1347, Z -3.8333, A 0.000, B 0.000, C 0.000 }
gfCNCPoint3[6864] = {X 258.4564, Y 48.8242, Z -3.8333, A 0.000, B 0.000, C 0.000 }
gfCNCPoint3[6865] = {X 257.6550, Y 48.3238, Z -3.8333, A 0.000, B 0.000, C 0.000 }
gfCNCPoint3[6866] = {X 256.9844, Y 47.6583, Z -3.8333, A 0.000, B 0.000, C 0.000 }
gfCNCPoint3[6867] = {X 256.4777, Y 46.8609, Z -3.8333, A 0.000, B 0.000, C 0.000 }
gfCNCPoint3[6868] = {X 256.1603, Y 45.9711, Z -3.8333, A 0.000, B 0.000, C 0.000 }
gfCNCPoint3[6869] = {X 256.0477, Y 45.0330, Z -3.8333, A 0.000, B 0.000, C 0.000 }
gfCNCPoint3[6870] = {X 256.0480, Y 44.1505, Z -3.8333, A 0.000, B 0.000, C 0.000 }
gfCNCPoint3[6871] = {X 256.1585, Y 43.2454, Z -3.8333, A 0.000, B 0.000, C 0.000 }
gfCNCPoint3[6872] = {X 256.4599, Y 42.3850, Z -3.8333, A 0.000, B 0.000, C 0.000 }
gfCNCPoint3[6873] = {X 256.9383, Y 41.6088, Z -3.8333, A 0.000, B 0.000, C 0.000 }
gfCNCPoint3[6874] = {X 257.5715, Y 40.9529, Z -3.8333, A 0.000, B 0.000, C 0.000 }
gfCNCPoint3[6875] = {X 257.5715, Y 34.3938, Z -3.8333, A 0.000, B 0.000, C 0.000 }
gfCNCPoint3[6876] = {X 254.7185, Y 34.3938, Z -3.8333, A 0.000, B 0.000, C 0.000 }
gfCNCPoint3[6877] = {X 250.3970, Y 42.8122, Z -3.8333, A 0.000, B 0.000, C 0.000 }
gfCNCPoint3[6878] = {X 250.5710, Y 43.4829, Z -3.8333, A 0.000, B 0.000, C 0.000 }
gfCNCPoint3[6879] = {X 250.6334, Y 44.1730, Z -3.8333, A 0.000, B 0.000, C 0.000 }
gfCNCPoint3[6880] = {X 250.6336, Y 45.0000, Z -3.8333, A 0.000, B 0.000, C 0.000 }
gfCNCPoint3[6881] = {X 250.5273, Y 45.9435, Z -3.8333, A 0.000, B 0.000, C 0.000 }
gfCNCPoint3[6882] = {X 250.2137, Y 46.8397, Z -3.8333, A 0.000, B 0.000, C 0.000 }
gfCNCPoint3[6883] = {X 249.7085, Y 47.6436, Z -3.8333, A 0.000, B 0.000, C 0.000 }
gfCNCPoint3[6884] = {X 249.0372, Y 48.3150, Z -3.8333, A 0.000, B 0.000, C 0.000 }
gfCNCPoint3[6885] = {X 248.2332, Y 48.8201, Z -3.8333, A 0.000, B 0.000, C 0.000 }
gfCNCPoint3[6886] = {X 247.3370, Y 49.1337, Z -3.8333, A 0.000, B 0.000, C 0.000 }
gfCNCPoint3[6887] = {X 246.3936, Y 49.2400, Z -3.8333, A 0.000, B 0.000, C 0.000 }
gfCNCPoint3[6888] = {X 239.8075, Y 49.2400, Z -3.8333, A 0.000, B 0.000, C 0.000 }
gfCNCPoint3[6889] = {X 238.8640, Y 49.1337, Z -3.8333, A 0.000, B 0.000, C 0.000 }
gfCNCPoint3[6890] = {X 237.9679, Y 48.8201, Z -3.8333, A 0.000, B 0.000, C 0.000 }
gfCNCPoint3[6891] = {X 237.1639, Y 48.3150, Z -3.8333, A 0.000, B 0.000, C 0.000 }
gfCNCPoint3[6892] = {X 236.4926, Y 47.6436, Z -3.8333, A 0.000, B 0.000, C 0.000 }
gfCNCPoint3[6893] = {X 235.9874, Y 46.8397, Z -3.8333, A 0.000, B 0.000, C 0.000 }
gfCNCPoint3[6894] = {X 235.6738, Y 45.9436, Z -3.8333, A 0.000, B 0.000, C 0.000 }
gfCNCPoint3[6895] = {X 235.5675, Y 45.0001, Z -3.8333, A 0.000, B 0.000, C 0.000 }
gfCNCPoint3[6896] = {X 235.5679, Y 44.1505, Z -3.8333, A 0.000, B 0.000, C 0.000 }
gfCNCPoint3[6897] = {X 235.6649, Y 43.3054, Z -3.8333, A 0.000, B 0.000, C 0.000 }
gfCNCPoint3[6898] = {X 235.9285, Y 42.4967, Z -3.8333, A 0.000, B 0.000, C 0.000 }
gfCNCPoint3[6899] = {X 236.3483, Y 41.7570, Z -3.8333, A 0.000, B 0.000, C 0.000 }
gfCNCPoint3[6900] = {X 236.9073, Y 41.1158, Z -3.8333, A 0.000, B 0.000, C 0.000 }
gfCNCPoint3[6901] = {X 237.5830, Y 40.5992, Z -3.8333, A 0.000, B 0.000, C 0.000 }
gfCNCPoint3[6902] = {X 238.3482, Y 40.2278, Z -3.8333, A 0.000, B 0.000, C 0.000 }
gfCNCPoint3[6903] = {X 242.3861, Y 32.3240, Z -3.8333, A 0.000, B 0.000, C 0.000 }
gfCNCPoint3[6904] = {X 241.2091, Y 31.5435, Z -3.8333, A 0.000, B 0.000, C 0.000 }
gfCNCPoint3[6905] = {X 240.1394, Y 30.6214, Z -3.8333, A 0.000, B 0.000, C 0.000 }
gfCNCPoint3[6906] = {X 239.1937, Y 29.5725, Z -3.8333, A 0.000, B 0.000, C 0.000 }
gfCNCPoint3[6907] = {X 238.3871, Y 28.4132, Z -3.8333, A 0.000, B 0.000, C 0.000 }
gfCNCPoint3[6908] = {X 237.7322, Y 27.1619, Z -3.8333, A 0.000, B 0.000, C 0.000 }
gfCNCPoint3[6909] = {X 237.2395, Y 25.8383, Z -3.8333, A 0.000, B 0.000, C 0.000 }
gfCNCPoint3[6910] = {X 236.8215, Y 24.0357, Z -3.8333, A 0.000, B 0.000, C 0.000 }
gfCNCPoint3[6911] = {X 236.6085, Y 22.1976, Z -3.8333, A 0.000, B 0.000, C 0.000 }
gfCNCPoint3[6912] = {X 236.6032, Y 20.3472, Z -3.8333, A 0.000, B 0.000, C 0.000 }
gfCNCPoint3[6913] = {X 236.8057, Y 18.5079, Z -3.8333, A 0.000, B 0.000, C 0.000 }
gfCNCPoint3[6914] = {X 237.2134, Y 16.7030, Z -3.8333, A 0.000, B 0.000, C 0.000 }
gfCNCPoint3[6915] = {X 237.7799, Y 15.1379, Z -3.8333, A 0.000, B 0.000, C 0.000 }
gfCNCPoint3[6916] = {X 238.5616, Y 13.6684, Z -3.8333, A 0.000, B 0.000, C 0.000 }
gfCNCPoint3[6917] = {X 239.5427, Y 12.3239, Z -3.8333, A 0.000, B 0.000, C 0.000 }
gfCNCPoint3[6918] = {X 240.7038, Y 11.1313, Z -3.8333, A 0.000, B 0.000, C 0.000 }
gfCNCPoint3[6919] = {X 242.0215, Y 10.1144, Z -3.8333, A 0.000, B 0.000, C 0.000 }
gfCNCPoint3[6920] = {X 243.4696, Y 9.2936, Z -3.8333, A 0.000, B 0.000, C 0.000 }
gfCNCPoint3[6921] = {X 245.0189, Y 8.6854, Z -3.8333, A 0.000, B 0.000, C 0.000 }
gfCNCPoint3[6922] = {X 246.6386, Y 8.3018, Z -3.8333, A 0.000, B 0.000, C 0.000 }
gfCNCPoint3[6923] = {X 248.7286, Y 8.0312, Z -3.8333, A 0.000, B 0.000, C 0.000 }
gfCNCPoint3[6924] = {X 250.8346, Y 7.9509, Z -3.8333, A 0.000, B 0.000, C 0.000 }
gfCNCPoint3[6925] = {X 266.7627, Y 7.9509, Z -3.8333, A 0.000, B 0.000, C 0.000 }
gfCNCPoint3[6926] = {X 267.7002, Y 8.0635, Z -3.8333, A 0.000, B 0.000, C 0.000 }
gfCNCPoint3[6927] = {X 268.5895, Y 8.3807, Z -3.8333, A 0.000, B 0.000, C 0.000 }
gfCNCPoint3[6928] = {X 269.3866, Y 8.8868, Z -3.8333, A 0.000, B 0.000, C 0.000 }
gfCNCPoint3[6929] = {X 270.0521, Y 9.5566, Z -3.8333, A 0.000, B 0.000, C 0.000 }
gfCNCPoint3[6930] = {X 270.5530, Y 10.3570, Z -3.8333, A 0.000, B 0.000, C 0.000 }
gfCNCPoint3[6931] = {X 270.8644, Y 11.2483, Z -3.8333, A 0.000, B 0.000, C 0.000 }
gfCNCPoint3[6932] = {X 270.9710, Y 12.1865, Z -3.8333, A 0.000, B 0.000, C 0.000 }
gfCNCPoint3[6933] = {X 270.9708, Y 13.0217, Z -3.8333, A 0.000, B 0.000, C 0.000 }
gfCNCPoint3[6934] = {X 270.8624, Y 13.9317, Z -3.8333, A 0.000, B 0.000, C 0.000 }
gfCNCPoint3[6935] = {X 270.5610, Y 14.7972, Z -3.8333, A 0.000, B 0.000, C 0.000 }
gfCNCPoint3[6936] = {X 270.0806, Y 15.5776, Z -3.8333, A 0.000, B 0.000, C 0.000 }
gfCNCPoint3[6937] = {X 269.4437, Y 16.2367, Z -3.8333, A 0.000, B 0.000, C 0.000 }
gfCNCPoint3[6938] = {X 269.4436, Y 28.5936, Z -3.8333, A 0.000, B 0.000, C 0.000 }
gfCNCPoint3[6939] = {X 273.4436, Y 28.5936, Z -3.8333, A 0.000, B 0.000, C 0.000 }
gfCNCPoint3[6940] = {X 269.3636, Y 28.5936, Z -3.8333, A 0.000, B 0.000, C 0.000 }
gfCNCPoint3[6941] = {X 269.3635, Y 40.9896, Z -3.8333, A 0.000, B 0.000, C 0.000 }
gfCNCPoint3[6942] = {X 269.4349, Y 41.0473, Z -3.8333, A 0.000, B 0.000, C 0.000 }
gfCNCPoint3[6943] = {X 270.0433, Y 41.6920, Z -3.8333, A 0.000, B 0.000, C 0.000 }
gfCNCPoint3[6944] = {X 270.5014, Y 42.4509, Z -3.8333, A 0.000, B 0.000, C 0.000 }
gfCNCPoint3[6945] = {X 270.7882, Y 43.2896, Z -3.8333, A 0.000, B 0.000, C 0.000 }
gfCNCPoint3[6946] = {X 270.8909, Y 44.1700, Z -3.8333, A 0.000, B 0.000, C 0.000 }
gfCNCPoint3[6947] = {X 270.8910, Y 45.0000, Z -3.8333, A 0.000, B 0.000, C 0.000 }
gfCNCPoint3[6948] = {X 270.7867, Y 45.9257, Z -3.8333, A 0.000, B 0.000, C 0.000 }
gfCNCPoint3[6949] = {X 270.4791, Y 46.8050, Z -3.8333, A 0.000, B 0.000, C 0.000 }
gfCNCPoint3[6950] = {X 269.9835, Y 47.5937, Z -3.8333, A 0.000, B 0.000, C 0.000 }
gfCNCPoint3[6951] = {X 269.3247, Y 48.2524, Z -3.8333, A 0.000, B 0.000, C 0.000 }
gfCNCPoint3[6952] = {X 268.5360, Y 48.7480, Z -3.8333, A 0.000, B 0.000, C 0.000 }
gfCNCPoint3[6953] = {X 267.6567, Y 49.0557, Z -3.8333, A 0.000, B 0.000, C 0.000 }
gfCNCPoint3[6954] = {X 266.7310, Y 49.1600, Z -3.8333, A 0.000, B 0.000, C 0.000 }
gfCNCPoint3[6955] = {X 260.2876, Y 49.1600, Z -3.8333, A 0.000, B 0.000, C 0.000 }
gfCNCPoint3[6956] = {X 259.3664, Y 49.0567, Z -3.8333, A 0.000, B 0.000, C 0.000 }
gfCNCPoint3[6957] = {X 258.4910, Y 48.7520, Z -3.8333, A 0.000, B 0.000, C 0.000 }
gfCNCPoint3[6958] = {X 257.7047, Y 48.2611, Z -3.8333, A 0.000, B 0.000, C 0.000 }
gfCNCPoint3[6959] = {X 257.0467, Y 47.6082, Z -3.8333, A 0.000, B 0.000, C 0.000 }
gfCNCPoint3[6960] = {X 256.5496, Y 46.8258, Z -3.8333, A 0.000, B 0.000, C 0.000 }
gfCNCPoint3[6961] = {X 256.2381, Y 45.9527, Z -3.8333, A 0.000, B 0.000, C 0.000 }
gfCNCPoint3[6962] = {X 256.1277, Y 45.0324, Z -3.8333, A 0.000, B 0.000, C 0.000 }
gfCNCPoint3[6963] = {X 256.1280, Y 44.1516, Z -3.8333, A 0.000, B 0.000, C 0.000 }
gfCNCPoint3[6964] = {X 256.2385, Y 43.2545, Z -3.8333, A 0.000, B 0.000, C 0.000 }
gfCNCPoint3[6965] = {X 256.5401, Y 42.4026, Z -3.8333, A 0.000, B 0.000, C 0.000 }
gfCNCPoint3[6966] = {X 257.0187, Y 41.6358, Z -3.8333, A 0.000, B 0.000, C 0.000 }
gfCNCPoint3[6967] = {X 257.6515, Y 40.9906, Z -3.8333, A 0.000, B 0.000, C 0.000 }
gfCNCPoint3[6968] = {X 257.6515, Y 34.3138, Z -3.8333, A 0.000, B 0.000, C 0.000 }
gfCNCPoint3[6969] = {X 254.6697, Y 34.3138, Z -3.8333, A 0.000, B 0.000, C 0.000 }
gfCNCPoint3[6970] = {X 250.3100, Y 42.8064, Z -3.8333, A 0.000, B 0.000, C 0.000 }
gfCNCPoint3[6971] = {X 250.4892, Y 43.4798, Z -3.8333, A 0.000, B 0.000, C 0.000 }
gfCNCPoint3[6972] = {X 250.5534, Y 44.1736, Z -3.8333, A 0.000, B 0.000, C 0.000 }
gfCNCPoint3[6973] = {X 250.5536, Y 45.0000, Z -3.8333, A 0.000, B 0.000, C 0.000 }
gfCNCPoint3[6974] = {X 250.4493, Y 45.9257, Z -3.8333, A 0.000, B 0.000, C 0.000 }
gfCNCPoint3[6975] = {X 250.1416, Y 46.8050, Z -3.8333, A 0.000, B 0.000, C 0.000 }
gfCNCPoint3[6976] = {X 249.6460, Y 47.5937, Z -3.8333, A 0.000, B 0.000, C 0.000 }
gfCNCPoint3[6977] = {X 248.9873, Y 48.2524, Z -3.8333, A 0.000, B 0.000, C 0.000 }
gfCNCPoint3[6978] = {X 248.1985, Y 48.7480, Z -3.8333, A 0.000, B 0.000, C 0.000 }
gfCNCPoint3[6979] = {X 247.3192, Y 49.0557, Z -3.8333, A 0.000, B 0.000, C 0.000 }
gfCNCPoint3[6980] = {X 246.3936, Y 49.1600, Z -3.8333, A 0.000, B 0.000, C 0.000 }
gfCNCPoint3[6981] = {X 239.8075, Y 49.1600, Z -3.8333, A 0.000, B 0.000, C 0.000 }
gfCNCPoint3[6982] = {X 238.8818, Y 49.0557, Z -3.8333, A 0.000, B 0.000, C 0.000 }
gfCNCPoint3[6983] = {X 238.0026, Y 48.7480, Z -3.8333, A 0.000, B 0.000, C 0.000 }
gfCNCPoint3[6984] = {X 237.2138, Y 48.2524, Z -3.8333, A 0.000, B 0.000, C 0.000 }
gfCNCPoint3[6985] = {X 236.5551, Y 47.5937, Z -3.8333, A 0.000, B 0.000, C 0.000 }
gfCNCPoint3[6986] = {X 236.0595, Y 46.8050, Z -3.8333, A 0.000, B 0.000, C 0.000 }
gfCNCPoint3[6987] = {X 235.7518, Y 45.9257, Z -3.8333, A 0.000, B 0.000, C 0.000 }
gfCNCPoint3[6988] = {X 235.6475, Y 45.0000, Z -3.8333, A 0.000, B 0.000, C 0.000 }
gfCNCPoint3[6989] = {X 235.6479, Y 44.1516, Z -3.8333, A 0.000, B 0.000, C 0.000 }
gfCNCPoint3[6990] = {X 235.7441, Y 43.3174, Z -3.8333, A 0.000, B 0.000, C 0.000 }
gfCNCPoint3[6991] = {X 236.0059, Y 42.5195, Z -3.8333, A 0.000, B 0.000, C 0.000 }
gfCNCPoint3[6992] = {X 236.4226, Y 41.7905, Z -3.8333, A 0.000, B 0.000, C 0.000 }
gfCNCPoint3[6993] = {X 236.9772, Y 41.1600, Z -3.8333, A 0.000, B 0.000, C 0.000 }
gfCNCPoint3[6994] = {X 237.6471, Y 40.6537, Z -3.8333, A 0.000, B 0.000, C 0.000 }
gfCNCPoint3[6995] = {X 238.4051, Y 40.2923, Z -3.8333, A 0.000, B 0.000, C 0.000 }
gfCNCPoint3[6996] = {X 242.4921, Y 32.2925, Z -3.8333, A 0.000, B 0.000, C 0.000 }
gfCNCPoint3[6997] = {X 241.3081, Y 31.5178, Z -3.8333, A 0.000, B 0.000, C 0.000 }
gfCNCPoint3[6998] = {X 240.2316, Y 30.5996, Z -3.8333, A 0.000, B 0.000, C 0.000 }
gfCNCPoint3[6999] = {X 239.2800, Y 29.5525, Z -3.8333, A 0.000, B 0.000, C 0.000 }
gfCNCPoint3[7000] = {X 238.4686, Y 28.3934, Z -3.8333, A 0.000, B 0.000, C 0.000 }
gfCNCPoint3[7001] = {X 237.8105, Y 27.1409, Z -3.8333, A 0.000, B 0.000, C 0.000 }
gfCNCPoint3[7002] = {X 237.3161, Y 25.8152, Z -3.8333, A 0.000, B 0.000, C 0.000 }
gfCNCPoint3[7003] = {X 236.9002, Y 24.0215, Z -3.8333, A 0.000, B 0.000, C 0.000 }
gfCNCPoint3[7004] = {X 236.6883, Y 22.1924, Z -3.8333, A 0.000, B 0.000, C 0.000 }
gfCNCPoint3[7005] = {X 236.6831, Y 20.3511, Z -3.8333, A 0.000, B 0.000, C 0.000 }
gfCNCPoint3[7006] = {X 236.8846, Y 18.5209, Z -3.8333, A 0.000, B 0.000, C 0.000 }
gfCNCPoint3[7007] = {X 237.2903, Y 16.7249, Z -3.8333, A 0.000, B 0.000, C 0.000 }
gfCNCPoint3[7008] = {X 237.8530, Y 15.1704, Z -3.8333, A 0.000, B 0.000, C 0.000 }
gfCNCPoint3[7009] = {X 238.6294, Y 13.7108, Z -3.8333, A 0.000, B 0.000, C 0.000 }
gfCNCPoint3[7010] = {X 239.6040, Y 12.3754, Z -3.8333, A 0.000, B 0.000, C 0.000 }
gfCNCPoint3[7011] = {X 240.7572, Y 11.1908, Z -3.8333, A 0.000, B 0.000, C 0.000 }
gfCNCPoint3[7012] = {X 242.0661, Y 10.1809, Z -3.8333, A 0.000, B 0.000, C 0.000 }
gfCNCPoint3[7013] = {X 243.5043, Y 9.3657, Z -3.8333, A 0.000, B 0.000, C 0.000 }
gfCNCPoint3[7014] = {X 245.0432, Y 8.7616, Z -3.8333, A 0.000, B 0.000, C 0.000 }
gfCNCPoint3[7015] = {X 246.6520, Y 8.3807, Z -3.8333, A 0.000, B 0.000, C 0.000 }
gfCNCPoint3[7016] = {X 248.7352, Y 8.1109, Z -3.8333, A 0.000, B 0.000, C 0.000 }
gfCNCPoint3[7017] = {X 250.8342, Y 8.0309, Z -3.8333, A 0.000, B 0.000, C 0.000 }
gfCNCPoint3[7018] = {X 266.7621, Y 8.0309, Z -3.8333, A 0.000, B 0.000, C 0.000 }
gfCNCPoint3[7019] = {X 267.6818, Y 8.1414, Z -3.8333, A 0.000, B 0.000, C 0.000 }
gfCNCPoint3[7020] = {X 268.5544, Y 8.4526, Z -3.8333, A 0.000, B 0.000, C 0.000 }
gfCNCPoint3[7021] = {X 269.3365, Y 8.9491, Z -3.8333, A 0.000, B 0.000, C 0.000 }
gfCNCPoint3[7022] = {X 269.9895, Y 9.6063, Z -3.8333, A 0.000, B 0.000, C 0.000 }
gfCNCPoint3[7023] = {X 270.4809, Y 10.3916, Z -3.8333, A 0.000, B 0.000, C 0.000 }
gfCNCPoint3[7024] = {X 270.7865, Y 11.2661, Z -3.8333, A 0.000, B 0.000, C 0.000 }
gfCNCPoint3[7025] = {X 270.8910, Y 12.1866, Z -3.8333, A 0.000, B 0.000, C 0.000 }
gfCNCPoint3[7026] = {X 270.8908, Y 13.0208, Z -3.8333, A 0.000, B 0.000, C 0.000 }
gfCNCPoint3[7027] = {X 270.7823, Y 13.9228, Z -3.8333, A 0.000, B 0.000, C 0.000 }
gfCNCPoint3[7028] = {X 270.4806, Y 14.7797, Z -3.8333, A 0.000, B 0.000, C 0.000 }
gfCNCPoint3[7029] = {X 270.0001, Y 15.5507, Z -3.8333, A 0.000, B 0.000, C 0.000 }
gfCNCPoint3[7030] = {X 269.3637, Y 16.1990, Z -3.8333, A 0.000, B 0.000, C 0.000 }
gfCNCPoint3[7031] = {X 269.3636, Y 28.5936, Z -3.8333, A 0.000, B 0.000, C 0.000 }
gfCNCPoint3[7032] = {X 273.3636, Y 28.5936, Z -3.8333, A 0.000, B 0.000, C 0.000 }
gfCNCPoint3[7033] = {X 269.2836, Y 28.5936, Z -3.8333, A 0.000, B 0.000, C 0.000 }
gfCNCPoint3[7034] = {X 269.2835, Y 41.0278, Z -3.8333, A 0.000, B 0.000, C 0.000 }
gfCNCPoint3[7035] = {X 269.3837, Y 41.1088, Z -3.8333, A 0.000, B 0.000, C 0.000 }
gfCNCPoint3[7036] = {X 269.9801, Y 41.7410, Z -3.8333, A 0.000, B 0.000, C 0.000 }
gfCNCPoint3[7037] = {X 270.4291, Y 42.4852, Z -3.8333, A 0.000, B 0.000, C 0.000 }
gfCNCPoint3[7038] = {X 270.7102, Y 43.3075, Z -3.8333, A 0.000, B 0.000, C 0.000 }
gfCNCPoint3[7039] = {X 270.8109, Y 44.1708, Z -3.8333, A 0.000, B 0.000, C 0.000 }
gfCNCPoint3[7040] = {X 270.8110, Y 45.0000, Z -3.8333, A 0.000, B 0.000, C 0.000 }
gfCNCPoint3[7041] = {X 270.7087, Y 45.9079, Z -3.8333, A 0.000, B 0.000, C 0.000 }
gfCNCPoint3[7042] = {X 270.4070, Y 46.7702, Z -3.8333, A 0.000, B 0.000, C 0.000 }
gfCNCPoint3[7043] = {X 269.9209, Y 47.5438, Z -3.8333, A 0.000, B 0.000, C 0.000 }
gfCNCPoint3[7044] = {X 269.2749, Y 48.1899, Z -3.8333, A 0.000, B 0.000, C 0.000 }
gfCNCPoint3[7045] = {X 268.5013, Y 48.6760, Z -3.8333, A 0.000, B 0.000, C 0.000 }
gfCNCPoint3[7046] = {X 267.6389, Y 48.9777, Z -3.8333, A 0.000, B 0.000, C 0.000 }
gfCNCPoint3[7047] = {X 266.7310, Y 49.0800, Z -3.8333, A 0.000, B 0.000, C 0.000 }
gfCNCPoint3[7048] = {X 260.2876, Y 49.0800, Z -3.8333, A 0.000, B 0.000, C 0.000 }
gfCNCPoint3[7049] = {X 259.3841, Y 48.9787, Z -3.8333, A 0.000, B 0.000, C 0.000 }
gfCNCPoint3[7050] = {X 258.5255, Y 48.6799, Z -3.8333, A 0.000, B 0.000, C 0.000 }
gfCNCPoint3[7051] = {X 257.7544, Y 48.1983, Z -3.8333, A 0.000, B 0.000, C 0.000 }
gfCNCPoint3[7052] = {X 257.1090, Y 47.5580, Z -3.8333, A 0.000, B 0.000, C 0.000 }
gfCNCPoint3[7053] = {X 256.6215, Y 46.7907, Z -3.8333, A 0.000, B 0.000, C 0.000 }
gfCNCPoint3[7054] = {X 256.3160, Y 45.9344, Z -3.8333, A 0.000, B 0.000, C 0.000 }
gfCNCPoint3[7055] = {X 256.2077, Y 45.0318, Z -3.8333, A 0.000, B 0.000, C 0.000 }
gfCNCPoint3[7056] = {X 256.2080, Y 44.1527, Z -3.8333, A 0.000, B 0.000, C 0.000 }
gfCNCPoint3[7057] = {X 256.3185, Y 43.2637, Z -3.8333, A 0.000, B 0.000, C 0.000 }
gfCNCPoint3[7058] = {X 256.6204, Y 42.4203, Z -3.8333, A 0.000, B 0.000, C 0.000 }
gfCNCPoint3[7059] = {X 257.0991, Y 41.6631, Z -3.8333, A 0.000, B 0.000, C 0.000 }
gfCNCPoint3[7060] = {X 257.7315, Y 41.0287, Z -3.8333, A 0.000, B 0.000, C 0.000 }
gfCNCPoint3[7061] = {X 257.7315, Y 34.2338, Z -3.8333, A 0.000, B 0.000, C 0.000 }
gfCNCPoint3[7062] = {X 254.6208, Y 34.2338, Z -3.8333, A 0.000, B 0.000, C 0.000 }
gfCNCPoint3[7063] = {X 250.2229, Y 42.8009, Z -3.8333, A 0.000, B 0.000, C 0.000 }
gfCNCPoint3[7064] = {X 250.4074, Y 43.4768, Z -3.8333, A 0.000, B 0.000, C 0.000 }
gfCNCPoint3[7065] = {X 250.4734, Y 44.1743, Z -3.8333, A 0.000, B 0.000, C 0.000 }
gfCNCPoint3[7066] = {X 250.4736, Y 45.0000, Z -3.8333, A 0.000, B 0.000, C 0.000 }
gfCNCPoint3[7067] = {X 250.3713, Y 45.9079, Z -3.8333, A 0.000, B 0.000, C 0.000 }
gfCNCPoint3[7068] = {X 250.0695, Y 46.7702, Z -3.8333, A 0.000, B 0.000, C 0.000 }
gfCNCPoint3[7069] = {X 249.5834, Y 47.5438, Z -3.8333, A 0.000, B 0.000, C 0.000 }
gfCNCPoint3[7070] = {X 248.9374, Y 48.1899, Z -3.8333, A 0.000, B 0.000, C 0.000 }
gfCNCPoint3[7071] = {X 248.1638, Y 48.6760, Z -3.8333, A 0.000, B 0.000, C 0.000 }
gfCNCPoint3[7072] = {X 247.3014, Y 48.9777, Z -3.8333, A 0.000, B 0.000, C 0.000 }
gfCNCPoint3[7073] = {X 246.3936, Y 49.0800, Z -3.8333, A 0.000, B 0.000, C 0.000 }
gfCNCPoint3[7074] = {X 239.8075, Y 49.0800, Z -3.8333, A 0.000, B 0.000, C 0.000 }
gfCNCPoint3[7075] = {X 238.8996, Y 48.9777, Z -3.8333, A 0.000, B 0.000, C 0.000 }
gfCNCPoint3[7076] = {X 238.0373, Y 48.6760, Z -3.8333, A 0.000, B 0.000, C 0.000 }
gfCNCPoint3[7077] = {X 237.2637, Y 48.1899, Z -3.8333, A 0.000, B 0.000, C 0.000 }
gfCNCPoint3[7078] = {X 236.6176, Y 47.5438, Z -3.8333, A 0.000, B 0.000, C 0.000 }
gfCNCPoint3[7079] = {X 236.1315, Y 46.7702, Z -3.8333, A 0.000, B 0.000, C 0.000 }
gfCNCPoint3[7080] = {X 235.8298, Y 45.9079, Z -3.8333, A 0.000, B 0.000, C 0.000 }
gfCNCPoint3[7081] = {X 235.7275, Y 45.0000, Z -3.8333, A 0.000, B 0.000, C 0.000 }
gfCNCPoint3[7082] = {X 235.7279, Y 44.1527, Z -3.8333, A 0.000, B 0.000, C 0.000 }
gfCNCPoint3[7083] = {X 235.8234, Y 43.3294, Z -3.8333, A 0.000, B 0.000, C 0.000 }
gfCNCPoint3[7084] = {X 236.0833, Y 42.5424, Z -3.8333, A 0.000, B 0.000, C 0.000 }
gfCNCPoint3[7085] = {X 236.4969, Y 41.8242, Z -3.8333, A 0.000, B 0.000, C 0.000 }
gfCNCPoint3[7086] = {X 237.0471, Y 41.2044, Z -3.8333, A 0.000, B 0.000, C 0.000 }
gfCNCPoint3[7087] = {X 237.7112, Y 40.7085, Z -3.8333, A 0.000, B 0.000, C 0.000 }
gfCNCPoint3[7088] = {X 238.4618, Y 40.3571, Z -3.8333, A 0.000, B 0.000, C 0.000 }
gfCNCPoint3[7089] = {X 242.5983, Y 32.2604, Z -3.8333, A 0.000, B 0.000, C 0.000 }
gfCNCPoint3[7090] = {X 241.4072, Y 31.4919, Z -3.8333, A 0.000, B 0.000, C 0.000 }
gfCNCPoint3[7091] = {X 240.3240, Y 30.5776, Z -3.8333, A 0.000, B 0.000, C 0.000 }
gfCNCPoint3[7092] = {X 239.3665, Y 29.5324, Z -3.8333, A 0.000, B 0.000, C 0.000 }
gfCNCPoint3[7093] = {X 238.5503, Y 28.3735, Z -3.8333, A 0.000, B 0.000, C 0.000 }
gfCNCPoint3[7094] = {X 237.8887, Y 27.1199, Z -3.8333, A 0.000, B 0.000, C 0.000 }
gfCNCPoint3[7095] = {X 237.3927, Y 25.7920, Z -3.8333, A 0.000, B 0.000, C 0.000 }
gfCNCPoint3[7096] = {X 236.9789, Y 24.0072, Z -3.8333, A 0.000, B 0.000, C 0.000 }
gfCNCPoint3[7097] = {X 236.7681, Y 22.1872, Z -3.8333, A 0.000, B 0.000, C 0.000 }
gfCNCPoint3[7098] = {X 236.7630, Y 20.3551, Z -3.8333, A 0.000, B 0.000, C 0.000 }
gfCNCPoint3[7099] = {X 236.9635, Y 18.5340, Z -3.8333, A 0.000, B 0.000, C 0.000 }
gfCNCPoint3[7100] = {X 237.3673, Y 16.7469, Z -3.8333, A 0.000, B 0.000, C 0.000 }
gfCNCPoint3[7101] = {X 237.9261, Y 15.2029, Z -3.8333, A 0.000, B 0.000, C 0.000 }
gfCNCPoint3[7102] = {X 238.6972, Y 13.7533, Z -3.8333, A 0.000, B 0.000, C 0.000 }
gfCNCPoint3[7103] = {X 239.6652, Y 12.4269, Z -3.8333, A 0.000, B 0.000, C 0.000 }
gfCNCPoint3[7104] = {X 240.8106, Y 11.2504, Z -3.8333, A 0.000, B 0.000, C 0.000 }
gfCNCPoint3[7105] = {X 242.1106, Y 10.2473, Z -3.8333, A 0.000, B 0.000, C 0.000 }
gfCNCPoint3[7106] = {X 243.5391, Y 9.4377, Z -3.8333, A 0.000, B 0.000, C 0.000 }
gfCNCPoint3[7107] = {X 245.0675, Y 8.8378, Z -3.8333, A 0.000, B 0.000, C 0.000 }
gfCNCPoint3[7108] = {X 246.6654, Y 8.4595, Z -3.8333, A 0.000, B 0.000, C 0.000 }
gfCNCPoint3[7109] = {X 248.7417, Y 8.1906, Z -3.8333, A 0.000, B 0.000, C 0.000 }
gfCNCPoint3[7110] = {X 250.8339, Y 8.1109, Z -3.8333, A 0.000, B 0.000, C 0.000 }
gfCNCPoint3[7111] = {X 266.7614, Y 8.1109, Z -3.8333, A 0.000, B 0.000, C 0.000 }
gfCNCPoint3[7112] = {X 267.6635, Y 8.2193, Z -3.8333, A 0.000, B 0.000, C 0.000 }
gfCNCPoint3[7113] = {X 268.5193, Y 8.5245, Z -3.8333, A 0.000, B 0.000, C 0.000 }
gfCNCPoint3[7114] = {X 269.2864, Y 9.0115, Z -3.8333, A 0.000, B 0.000, C 0.000 }
gfCNCPoint3[7115] = {X 269.9268, Y 9.6560, Z -3.8333, A 0.000, B 0.000, C 0.000 }
gfCNCPoint3[7116] = {X 270.4088, Y 10.4262, Z -3.8333, A 0.000, B 0.000, C 0.000 }
gfCNCPoint3[7117] = {X 270.7085, Y 11.2840, Z -3.8333, A 0.000, B 0.000, C 0.000 }
gfCNCPoint3[7118] = {X 270.8110, Y 12.1867, Z -3.8333, A 0.000, B 0.000, C 0.000 }
gfCNCPoint3[7119] = {X 270.8108, Y 13.0200, Z -3.8333, A 0.000, B 0.000, C 0.000 }
gfCNCPoint3[7120] = {X 270.7023, Y 13.9138, Z -3.8333, A 0.000, B 0.000, C 0.000 }
gfCNCPoint3[7121] = {X 270.4003, Y 14.7621, Z -3.8333, A 0.000, B 0.000, C 0.000 }
gfCNCPoint3[7122] = {X 269.9197, Y 15.5234, Z -3.8333, A 0.000, B 0.000, C 0.000 }
gfCNCPoint3[7123] = {X 269.2837, Y 16.1608, Z -3.8333, A 0.000, B 0.000, C 0.000 }
gfCNCPoint3[7124] = {X 269.2836, Y 28.5936, Z -3.8333, A 0.000, B 0.000, C 0.000 }
gfCNCPoint3[7125] = {X 273.2836, Y 28.5936, Z -3.8333, A 0.000, B 0.000, C 0.000 }
gfCNCPoint3[7126] = {X 269.2036, Y 28.5936, Z -3.8333, A 0.000, B 0.000, C 0.000 }
gfCNCPoint3[7127] = {X 269.2035, Y 41.0659, Z -3.8333, A 0.000, B 0.000, C 0.000 }
gfCNCPoint3[7128] = {X 269.3424, Y 41.1788, Z -3.8333, A 0.000, B 0.000, C 0.000 }
gfCNCPoint3[7129] = {X 269.9284, Y 41.8053, Z -3.8333, A 0.000, B 0.000, C 0.000 }
gfCNCPoint3[7130] = {X 270.3674, Y 42.5423, Z -3.8333, A 0.000, B 0.000, C 0.000 }
gfCNCPoint3[7131] = {X 270.6391, Y 43.3560, Z -3.8333, A 0.000, B 0.000, C 0.000 }
gfCNCPoint3[7132] = {X 270.7310, Y 44.2089, Z -3.8333, A 0.000, B 0.000, C 0.000 }
gfCNCPoint3[7133] = {X 270.7310, Y 45.0000, Z -3.8333, A 0.000, B 0.000, C 0.000 }
gfCNCPoint3[7134] = {X 270.6307, Y 45.8901, Z -3.8333, A 0.000, B 0.000, C 0.000 }
gfCNCPoint3[7135] = {X 270.3349, Y 46.7355, Z -3.8333, A 0.000, B 0.000, C 0.000 }
gfCNCPoint3[7136] = {X 269.8584, Y 47.4940, Z -3.8333, A 0.000, B 0.000, C 0.000 }
gfCNCPoint3[7137] = {X 269.2250, Y 48.1273, Z -3.8333, A 0.000, B 0.000, C 0.000 }
gfCNCPoint3[7138] = {X 268.4666, Y 48.6039, Z -3.8333, A 0.000, B 0.000, C 0.000 }
gfCNCPoint3[7139] = {X 267.6211, Y 48.8997, Z -3.8333, A 0.000, B 0.000, C 0.000 }
gfCNCPoint3[7140] = {X 266.7310, Y 49.0000, Z -3.8333, A 0.000, B 0.000, C 0.000 }
gfCNCPoint3[7141] = {X 260.2876, Y 49.0000, Z -3.8333, A 0.000, B 0.000, C 0.000 }
gfCNCPoint3[7142] = {X 259.3975, Y 48.8997, Z -3.8333, A 0.000, B 0.000, C 0.000 }
gfCNCPoint3[7143] = {X 258.5520, Y 48.6039, Z -3.8333, A 0.000, B 0.000, C 0.000 }
gfCNCPoint3[7144] = {X 257.7936, Y 48.1273, Z -3.8333, A 0.000, B 0.000, C 0.000 }
gfCNCPoint3[7145] = {X 257.1602, Y 47.4939, Z -3.8333, A 0.000, B 0.000, C 0.000 }
gfCNCPoint3[7146] = {X 256.6837, Y 46.7355, Z -3.8333, A 0.000, B 0.000, C 0.000 }
gfCNCPoint3[7147] = {X 256.3878, Y 45.8901, Z -3.8333, A 0.000, B 0.000, C 0.000 }
gfCNCPoint3[7148] = {X 256.2876, Y 45.0000, Z -3.8333, A 0.000, B 0.000, C 0.000 }
gfCNCPoint3[7149] = {X 256.2879, Y 44.1538, Z -3.8333, A 0.000, B 0.000, C 0.000 }
gfCNCPoint3[7150] = {X 256.3986, Y 43.2730, Z -3.8333, A 0.000, B 0.000, C 0.000 }
gfCNCPoint3[7151] = {X 256.7008, Y 42.4382, Z -3.8333, A 0.000, B 0.000, C 0.000 }
gfCNCPoint3[7152] = {X 257.1796, Y 41.6907, Z -3.8333, A 0.000, B 0.000, C 0.000 }
gfCNCPoint3[7153] = {X 257.8115, Y 41.0672, Z -3.8333, A 0.000, B 0.000, C 0.000 }
gfCNCPoint3[7154] = {X 257.8115, Y 34.1538, Z -3.8333, A 0.000, B 0.000, C 0.000 }
gfCNCPoint3[7155] = {X 254.8162, Y 34.1538, Z -3.8333, A 0.000, B 0.000, C 0.000 }
gfCNCPoint3[7156] = {X 254.5729, Y 34.1520, Z -3.8333, A 0.000, B 0.000, C 0.000 }
gfCNCPoint3[7157] = {X 250.1357, Y 42.7958, Z -3.8333, A 0.000, B 0.000, C 0.000 }
gfCNCPoint3[7158] = {X 250.3286, Y 43.4907, Z -3.8333, A 0.000, B 0.000, C 0.000 }
gfCNCPoint3[7159] = {X 250.3936, Y 44.2089, Z -3.8333, A 0.000, B 0.000, C 0.000 }
gfCNCPoint3[7160] = {X 250.3936, Y 45.0000, Z -3.8333, A 0.000, B 0.000, C 0.000 }
gfCNCPoint3[7161] = {X 250.2933, Y 45.8901, Z -3.8333, A 0.000, B 0.000, C 0.000 }
gfCNCPoint3[7162] = {X 249.9974, Y 46.7355, Z -3.8333, A 0.000, B 0.000, C 0.000 }
gfCNCPoint3[7163] = {X 249.5209, Y 47.4940, Z -3.8333, A 0.000, B 0.000, C 0.000 }
gfCNCPoint3[7164] = {X 248.8875, Y 48.1273, Z -3.8333, A 0.000, B 0.000, C 0.000 }
gfCNCPoint3[7165] = {X 248.1291, Y 48.6039, Z -3.8333, A 0.000, B 0.000, C 0.000 }
gfCNCPoint3[7166] = {X 247.2836, Y 48.8997, Z -3.8333, A 0.000, B 0.000, C 0.000 }
gfCNCPoint3[7167] = {X 246.3936, Y 49.0000, Z -3.8333, A 0.000, B 0.000, C 0.000 }
gfCNCPoint3[7168] = {X 239.8075, Y 49.0000, Z -3.8333, A 0.000, B 0.000, C 0.000 }
gfCNCPoint3[7169] = {X 238.9174, Y 48.8997, Z -3.8333, A 0.000, B 0.000, C 0.000 }
gfCNCPoint3[7170] = {X 238.0720, Y 48.6039, Z -3.8333, A 0.000, B 0.000, C 0.000 }
gfCNCPoint3[7171] = {X 237.3135, Y 48.1273, Z -3.8333, A 0.000, B 0.000, C 0.000 }
gfCNCPoint3[7172] = {X 236.6802, Y 47.4940, Z -3.8333, A 0.000, B 0.000, C 0.000 }
gfCNCPoint3[7173] = {X 236.2036, Y 46.7355, Z -3.8333, A 0.000, B 0.000, C 0.000 }
gfCNCPoint3[7174] = {X 235.9078, Y 45.8901, Z -3.8333, A 0.000, B 0.000, C 0.000 }
gfCNCPoint3[7175] = {X 235.8075, Y 45.0000, Z -3.8333, A 0.000, B 0.000, C 0.000 }
gfCNCPoint3[7176] = {X 235.8079, Y 44.1538, Z -3.8333, A 0.000, B 0.000, C 0.000 }
gfCNCPoint3[7177] = {X 235.9027, Y 43.3414, Z -3.8333, A 0.000, B 0.000, C 0.000 }
gfCNCPoint3[7178] = {X 236.1607, Y 42.5654, Z -3.8333, A 0.000, B 0.000, C 0.000 }
gfCNCPoint3[7179] = {X 236.5712, Y 41.8580, Z -3.8333, A 0.000, B 0.000, C 0.000 }
gfCNCPoint3[7180] = {X 237.1169, Y 41.2489, Z -3.8333, A 0.000, B 0.000, C 0.000 }
gfCNCPoint3[7181] = {X 237.7752, Y 40.7635, Z -3.8333, A 0.000, B 0.000, C 0.000 }
gfCNCPoint3[7182] = {X 238.5184, Y 40.4222, Z -3.8333, A 0.000, B 0.000, C 0.000 }
gfCNCPoint3[7183] = {X 242.7047, Y 32.2279, Z -3.8333, A 0.000, B 0.000, C 0.000 }
gfCNCPoint3[7184] = {X 241.5066, Y 31.4657, Z -3.8333, A 0.000, B 0.000, C 0.000 }
gfCNCPoint3[7185] = {X 240.4166, Y 30.5554, Z -3.8333, A 0.000, B 0.000, C 0.000 }
gfCNCPoint3[7186] = {X 239.4530, Y 29.5123, Z -3.8333, A 0.000, B 0.000, C 0.000 }
gfCNCPoint3[7187] = {X 238.6319, Y 28.3536, Z -3.8333, A 0.000, B 0.000, C 0.000 }
gfCNCPoint3[7188] = {X 237.9670, Y 27.0989, Z -3.8333, A 0.000, B 0.000, C 0.000 }
gfCNCPoint3[7189] = {X 237.4692, Y 25.7689, Z -3.8333, A 0.000, B 0.000, C 0.000 }
gfCNCPoint3[7190] = {X 237.0576, Y 23.9929, Z -3.8333, A 0.000, B 0.000, C 0.000 }
gfCNCPoint3[7191] = {X 236.8480, Y 22.1820, Z -3.8333, A 0.000, B 0.000, C 0.000 }
gfCNCPoint3[7192] = {X 236.8429, Y 20.3590, Z -3.8333, A 0.000, B 0.000, C 0.000 }
gfCNCPoint3[7193] = {X 237.0425, Y 18.5469, Z -3.8333, A 0.000, B 0.000, C 0.000 }
gfCNCPoint3[7194] = {X 237.4442, Y 16.7687, Z -3.8333, A 0.000, B 0.000, C 0.000 }
gfCNCPoint3[7195] = {X 237.9992, Y 15.2354, Z -3.8333, A 0.000, B 0.000, C 0.000 }
gfCNCPoint3[7196] = {X 238.7651, Y 13.7956, Z -3.8333, A 0.000, B 0.000, C 0.000 }
gfCNCPoint3[7197] = {X 239.7264, Y 12.4784, Z -3.8333, A 0.000, B 0.000, C 0.000 }
gfCNCPoint3[7198] = {X 240.8640, Y 11.3100, Z -3.8333, A 0.000, B 0.000, C 0.000 }
gfCNCPoint3[7199] = {X 242.1551, Y 10.3138, Z -3.8333, A 0.000, B 0.000, C 0.000 }
gfCNCPoint3[7200] = {X 243.5738, Y 9.5098, Z -3.8333, A 0.000, B 0.000, C 0.000 }
gfCNCPoint3[7201] = {X 245.0918, Y 8.9140, Z -3.8333, A 0.000, B 0.000, C 0.000 }
gfCNCPoint3[7202] = {X 246.6787, Y 8.5384, Z -3.8333, A 0.000, B 0.000, C 0.000 }
gfCNCPoint3[7203] = {X 248.7483, Y 8.2704, Z -3.8333, A 0.000, B 0.000, C 0.000 }
gfCNCPoint3[7204] = {X 250.8336, Y 8.1909, Z -3.8333, A 0.000, B 0.000, C 0.000 }
gfCNCPoint3[7205] = {X 266.7608, Y 8.1909, Z -3.8333, A 0.000, B 0.000, C 0.000 }
gfCNCPoint3[7206] = {X 267.6452, Y 8.2972, Z -3.8333, A 0.000, B 0.000, C 0.000 }
gfCNCPoint3[7207] = {X 268.4842, Y 8.5964, Z -3.8333, A 0.000, B 0.000, C 0.000 }
gfCNCPoint3[7208] = {X 269.2363, Y 9.0738, Z -3.8333, A 0.000, B 0.000, C 0.000 }
gfCNCPoint3[7209] = {X 269.8641, Y 9.7057, Z -3.8333, A 0.000, B 0.000, C 0.000 }
gfCNCPoint3[7210] = {X 270.3367, Y 10.4608, Z -3.8333, A 0.000, B 0.000, C 0.000 }
gfCNCPoint3[7211] = {X 270.6305, Y 11.3018, Z -3.8333, A 0.000, B 0.000, C 0.000 }
gfCNCPoint3[7212] = {X 270.7310, Y 12.1869, Z -3.8333, A 0.000, B 0.000, C 0.000 }
gfCNCPoint3[7213] = {X 270.7308, Y 13.0192, Z -3.8333, A 0.000, B 0.000, C 0.000 }
gfCNCPoint3[7214] = {X 270.6222, Y 13.9048, Z -3.8333, A 0.000, B 0.000, C 0.000 }
gfCNCPoint3[7215] = {X 270.3200, Y 14.7443, Z -3.8333, A 0.000, B 0.000, C 0.000 }
gfCNCPoint3[7216] = {X 269.8392, Y 15.4959, Z -3.8333, A 0.000, B 0.000, C 0.000 }
gfCNCPoint3[7217] = {X 269.2037, Y 16.1222, Z -3.8333, A 0.000, B 0.000, C 0.000 }
gfCNCPoint3[7218] = {X 269.2036, Y 28.5936, Z -3.8333, A 0.000, B 0.000, C 0.000 }
gfCNCPoint3[7219] = {X 273.2836, Y 28.5936, Z -3.8333, A 0.000, B 0.000, C 0.000 }
gfCNCPoint3[7220] = {X 273.2836, Y 28.5936, Z -0.8333, A 0.000, B 0.000, C 0.000 }
gfCNCPoint3[7221] = {X 273.2836, Y 28.5936, Z 11.0000, A 0.000, B 0.000, C 0.000 }
gfCNCPoint3[7222] = {X 277.7454, Y 28.5927, Z 11.0000, A 0.000, B 0.000, C 0.000 }
gfCNCPoint3[7223] = {X 277.7454, Y 28.5927, Z -0.8333, A 0.000, B 0.000, C 0.000 }
gfCNCPoint3[7224] = {X 277.7454, Y 28.5927, Z -3.8333, A 0.000, B 0.000, C 0.000 }
gfCNCPoint3[7225] = {X 281.8254, Y 28.5926, Z -3.8333, A 0.000, B 0.000, C 0.000 }
gfCNCPoint3[7226] = {X 281.8252, Y 16.2742, Z -3.8333, A 0.000, B 0.000, C 0.000 }
gfCNCPoint3[7227] = {X 281.1867, Y 15.6031, Z -3.8333, A 0.000, B 0.000, C 0.000 }
gfCNCPoint3[7228] = {X 280.7059, Y 14.8113, Z -3.8333, A 0.000, B 0.000, C 0.000 }
gfCNCPoint3[7229] = {X 280.4050, Y 13.9352, Z -3.8333, A 0.000, B 0.000, C 0.000 }
gfCNCPoint3[7230] = {X 280.2978, Y 13.0151, Z -3.8333, A 0.000, B 0.000, C 0.000 }
gfCNCPoint3[7231] = {X 280.2977, Y 12.1868, Z -3.8333, A 0.000, B 0.000, C 0.000 }
gfCNCPoint3[7232] = {X 280.4060, Y 11.2255, Z -3.8333, A 0.000, B 0.000, C 0.000 }
gfCNCPoint3[7233] = {X 280.7255, Y 10.3124, Z -3.8333, A 0.000, B 0.000, C 0.000 }
gfCNCPoint3[7234] = {X 281.2402, Y 9.4933, Z -3.8333, A 0.000, B 0.000, C 0.000 }
gfCNCPoint3[7235] = {X 281.9242, Y 8.8093, Z -3.8333, A 0.000, B 0.000, C 0.000 }
gfCNCPoint3[7236] = {X 282.7433, Y 8.2946, Z -3.8333, A 0.000, B 0.000, C 0.000 }
gfCNCPoint3[7237] = {X 283.6564, Y 7.9751, Z -3.8333, A 0.000, B 0.000, C 0.000 }
gfCNCPoint3[7238] = {X 284.6177, Y 7.8668, Z -3.8333, A 0.000, B 0.000, C 0.000 }
gfCNCPoint3[7239] = {X 291.0611, Y 7.8668, Z -3.8333, A 0.000, B 0.000, C 0.000 }
gfCNCPoint3[7240] = {X 292.0224, Y 7.9751, Z -3.8333, A 0.000, B 0.000, C 0.000 }
gfCNCPoint3[7241] = {X 292.9355, Y 8.2946, Z -3.8333, A 0.000, B 0.000, C 0.000 }
gfCNCPoint3[7242] = {X 293.7546, Y 8.8093, Z -3.8333, A 0.000, B 0.000, C 0.000 }
gfCNCPoint3[7243] = {X 294.4386, Y 9.4933, Z -3.8333, A 0.000, B 0.000, C 0.000 }
gfCNCPoint3[7244] = {X 294.9533, Y 10.3124, Z -3.8333, A 0.000, B 0.000, C 0.000 }
gfCNCPoint3[7245] = {X 295.2728, Y 11.2255, Z -3.8333, A 0.000, B 0.000, C 0.000 }
gfCNCPoint3[7246] = {X 295.3811, Y 12.1868, Z -3.8333, A 0.000, B 0.000, C 0.000 }
gfCNCPoint3[7247] = {X 295.3811, Y 12.9782, Z -3.8333, A 0.000, B 0.000, C 0.000 }
gfCNCPoint3[7248] = {X 295.2797, Y 13.9081, Z -3.8333, A 0.000, B 0.000, C 0.000 }
gfCNCPoint3[7249] = {X 294.9805, Y 14.7945, Z -3.8333, A 0.000, B 0.000, C 0.000 }
gfCNCPoint3[7250] = {X 294.4975, Y 15.5956, Z -3.8333, A 0.000, B 0.000, C 0.000 }
gfCNCPoint3[7251] = {X 293.8533, Y 16.2740, Z -3.8333, A 0.000, B 0.000, C 0.000 }
gfCNCPoint3[7252] = {X 293.8545, Y 22.1965, Z -3.8333, A 0.000, B 0.000, C 0.000 }
gfCNCPoint3[7253] = {X 302.7594, Y 22.1965, Z -3.8333, A 0.000, B 0.000, C 0.000 }
gfCNCPoint3[7254] = {X 302.7642, Y 16.2779, Z -3.8333, A 0.000, B 0.000, C 0.000 }
gfCNCPoint3[7255] = {X 302.1242, Y 15.6068, Z -3.8333, A 0.000, B 0.000, C 0.000 }
gfCNCPoint3[7256] = {X 301.6421, Y 14.8146, Z -3.8333, A 0.000, B 0.000, C 0.000 }
gfCNCPoint3[7257] = {X 301.3402, Y 13.9377, Z -3.8333, A 0.000, B 0.000, C 0.000 }
gfCNCPoint3[7258] = {X 301.2324, Y 13.0165, Z -3.8333, A 0.000, B 0.000, C 0.000 }
gfCNCPoint3[7259] = {X 301.2323, Y 12.1868, Z -3.8333, A 0.000, B 0.000, C 0.000 }
gfCNCPoint3[7260] = {X 301.3406, Y 11.2255, Z -3.8333, A 0.000, B 0.000, C 0.000 }
gfCNCPoint3[7261] = {X 301.6601, Y 10.3124, Z -3.8333, A 0.000, B 0.000, C 0.000 }
gfCNCPoint3[7262] = {X 302.1747, Y 9.4933, Z -3.8333, A 0.000, B 0.000, C 0.000 }
gfCNCPoint3[7263] = {X 302.8588, Y 8.8093, Z -3.8333, A 0.000, B 0.000, C 0.000 }
gfCNCPoint3[7264] = {X 303.6779, Y 8.2946, Z -3.8333, A 0.000, B 0.000, C 0.000 }
gfCNCPoint3[7265] = {X 304.5910, Y 7.9751, Z -3.8333, A 0.000, B 0.000, C 0.000 }
gfCNCPoint3[7266] = {X 305.5523, Y 7.8668, Z -3.8333, A 0.000, B 0.000, C 0.000 }
gfCNCPoint3[7267] = {X 311.9957, Y 7.8668, Z -3.8333, A 0.000, B 0.000, C 0.000 }
gfCNCPoint3[7268] = {X 312.9570, Y 7.9751, Z -3.8333, A 0.000, B 0.000, C 0.000 }
gfCNCPoint3[7269] = {X 313.8701, Y 8.2946, Z -3.8333, A 0.000, B 0.000, C 0.000 }
